Yaskawa INFORM job: DEMO_ROOF_SIDE_0625_3PAINT_47.JBI

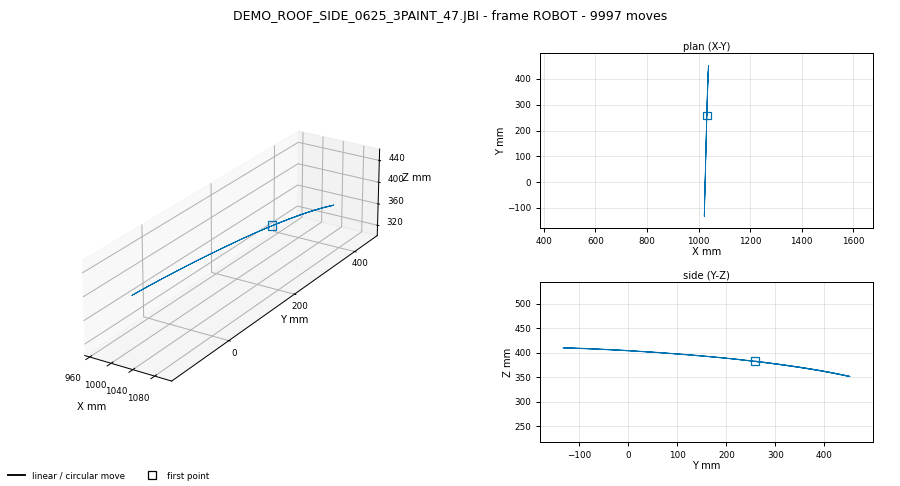
[picture p0: tool path of DEMO_ROOF_SIDE_0625_3PAINT_47.JBI in frame ROBOT, 9997 of 9997 moves have a stored position in this frame; points joined in program order, loops and branches not executed]
/JOB
//NAME DEMO_ROOF_SIDE_0625_3PAINT47
//POS
///NPOS 9997,0,0,0,0,0
///TOOL 0
///USER 0
///POSTYPE ROBOT
///RECTAN
///RCONF 1,0,0,0,0,0,0,0,0,0,0,0,0,0,0,0,0,0,0,0,0,0,0,0
C00000=1032.456,258.256,382.887,170.687,44.569,158.534
C00001=1032.463,258.505,382.858,170.690,44.569,158.534
C00002=1032.469,258.753,382.828,170.693,44.568,158.534
C00003=1032.477,259.001,382.799,170.697,44.568,158.535
C00004=1032.483,259.249,382.770,170.701,44.568,158.535
C00005=1032.490,259.497,382.740,170.704,44.568,158.535
C00006=1032.497,259.745,382.710,170.707,44.567,158.535
C00007=1032.504,259.994,382.681,170.711,44.567,158.536
C00008=1032.510,260.241,382.651,170.714,44.567,158.536
C00009=1032.517,260.490,382.621,170.718,44.567,158.536
C00010=1032.525,260.738,382.592,170.721,44.567,158.537
C00011=1032.531,260.986,382.563,170.725,44.566,158.537
C00012=1032.538,261.234,382.533,170.728,44.566,158.537
C00013=1032.545,261.482,382.503,170.731,44.566,158.537
C00014=1032.552,261.730,382.473,170.734,44.566,158.538
C00015=1032.558,261.979,382.444,170.739,44.566,158.538
C00016=1032.565,262.227,382.414,170.742,44.566,158.538
C00017=1032.572,262.475,382.383,170.745,44.566,158.539
C00018=1032.581,262.826,382.341,170.749,44.566,158.539
C00019=1032.590,263.179,382.299,170.755,44.566,158.540
C00020=1032.600,263.530,382.256,170.759,44.566,158.540
C00021=1032.609,263.882,382.214,170.765,44.566,158.541
C00022=1032.616,264.130,382.183,170.768,44.566,158.541
C00023=1032.623,264.378,382.154,170.771,44.566,158.541
C00024=1032.630,264.626,382.124,170.775,44.566,158.541
C00025=1032.636,264.875,382.093,170.779,44.566,158.542
C00026=1032.643,265.122,382.063,170.782,44.566,158.542
C00027=1032.650,265.370,382.033,170.786,44.566,158.542
C00028=1032.656,265.619,382.003,170.789,44.566,158.543
C00029=1032.662,265.867,381.973,170.792,44.566,158.543
C00030=1032.670,266.115,381.943,170.796,44.565,158.543
C00031=1032.677,266.363,381.913,170.800,44.565,158.544
C00032=1032.683,266.611,381.883,170.803,44.565,158.544
C00033=1032.690,266.859,381.852,170.806,44.565,158.544
C00034=1032.697,267.108,381.822,170.810,44.565,158.545
C00035=1032.703,267.355,381.792,170.814,44.565,158.545
C00036=1032.710,267.604,381.762,170.817,44.565,158.545
C00037=1032.717,267.851,381.731,170.821,44.566,158.546
C00038=1032.723,268.099,381.701,170.824,44.566,158.546
C00039=1032.730,268.347,381.671,170.828,44.565,158.546
C00040=1032.737,268.596,381.640,170.831,44.565,158.547
C00041=1032.743,268.843,381.610,170.835,44.565,158.547
C00042=1032.750,269.092,381.579,170.838,44.565,158.547
C00043=1032.757,269.340,381.549,170.842,44.566,158.548
C00044=1032.764,269.588,381.519,170.846,44.566,158.548
C00045=1032.770,269.835,381.488,170.849,44.566,158.549
C00046=1032.777,270.084,381.458,170.852,44.566,158.549
C00047=1032.784,270.332,381.427,170.856,44.566,158.549
C00048=1032.791,270.580,381.397,170.860,44.566,158.549
C00049=1032.797,270.828,381.366,170.864,44.566,158.550
C00050=1032.804,271.076,381.336,170.867,44.566,158.550
C00051=1032.811,271.324,381.305,170.870,44.566,158.551
C00052=1032.818,271.573,381.275,170.874,44.566,158.551
C00053=1032.824,271.820,381.244,170.878,44.567,158.551
C00054=1032.831,272.068,381.214,170.881,44.566,158.552
C00055=1032.837,272.317,381.183,170.885,44.566,158.552
C00056=1032.844,272.564,381.152,170.889,44.567,158.553
C00057=1032.851,272.812,381.122,170.892,44.567,158.553
C00058=1032.857,273.060,381.091,170.896,44.567,158.553
C00059=1032.865,273.308,381.060,170.900,44.567,158.554
C00060=1032.871,273.557,381.030,170.903,44.567,158.554
C00061=1032.878,273.804,380.998,170.907,44.567,158.554
C00062=1032.884,274.052,380.969,170.910,44.568,158.555
C00063=1032.891,274.300,380.937,170.914,44.568,158.555
C00064=1032.897,274.548,380.906,170.918,44.568,158.555
C00065=1032.905,274.796,380.876,170.921,44.568,158.556
C00066=1032.911,275.045,380.845,170.926,44.568,158.556
C00067=1032.918,275.292,380.813,170.929,44.568,158.557
C00068=1032.925,275.540,380.784,170.932,44.569,158.557
C00069=1032.931,275.788,380.752,170.936,44.569,158.557
C00070=1032.938,276.036,380.721,170.940,44.569,158.558
C00071=1032.945,276.284,380.691,170.943,44.569,158.558
C00072=1032.952,276.532,380.659,170.947,44.569,158.558
C00073=1032.958,276.780,380.628,170.951,44.569,158.559
C00074=1032.969,277.137,380.585,170.957,44.569,158.560
C00075=1032.978,277.493,380.540,170.961,44.570,158.560
C00076=1032.988,277.850,380.495,170.967,44.570,158.561
C00077=1032.997,278.206,380.451,170.972,44.570,158.561
C00078=1033.004,278.453,380.419,170.976,44.571,158.562
C00079=1033.011,278.702,380.388,170.980,44.571,158.562
C00080=1033.017,278.950,380.357,170.984,44.571,158.562
C00081=1033.024,279.198,380.326,170.987,44.571,158.563
C00082=1033.031,279.446,380.294,170.992,44.572,158.563
C00083=1033.037,279.694,380.263,170.995,44.572,158.564
C00084=1033.044,279.942,380.232,170.998,44.572,158.564
C00085=1033.051,280.190,380.201,171.003,44.573,158.565
C00086=1033.058,280.438,380.170,171.006,44.573,158.565
C00087=1033.065,280.686,380.138,171.010,44.573,158.565
C00088=1033.071,280.933,380.107,171.014,44.573,158.566
C00089=1033.078,281.181,380.075,171.018,44.574,158.566
C00090=1033.085,281.429,380.044,171.021,44.574,158.567
C00091=1033.092,281.677,380.013,171.025,44.574,158.567
C00092=1033.098,281.925,379.981,171.029,44.575,158.568
C00093=1033.105,282.173,379.950,171.032,44.575,158.568
C00094=1033.112,282.421,379.918,171.037,44.575,158.568
C00095=1033.119,282.669,379.887,171.040,44.576,158.569
C00096=1033.125,282.917,379.855,171.045,44.575,158.569
C00097=1033.132,283.165,379.824,171.048,44.576,158.570
C00098=1033.139,283.412,379.793,171.052,44.577,158.570
C00099=1033.145,283.660,379.761,171.056,44.576,158.570
C00100=1033.153,283.908,379.730,171.059,44.577,158.571
C00101=1033.160,284.156,379.699,171.064,44.577,158.571
C00102=1033.166,284.404,379.667,171.067,44.578,158.572
C00103=1033.173,284.652,379.636,171.071,44.578,158.572
C00104=1033.180,284.900,379.605,171.075,44.578,158.573
C00105=1033.187,285.147,379.573,171.079,44.579,158.573
C00106=1033.194,285.396,379.541,171.083,44.579,158.574
C00107=1033.201,285.644,379.510,171.087,44.579,158.574
C00108=1033.208,285.891,379.478,171.091,44.580,158.575
C00109=1033.214,286.139,379.446,171.094,44.580,158.575
C00110=1033.221,286.387,379.415,171.098,44.580,158.575
C00111=1033.228,286.635,379.383,171.102,44.581,158.576
C00112=1033.235,286.883,379.352,171.106,44.581,158.576
C00113=1033.241,287.130,379.319,171.111,44.582,158.577
C00114=1033.248,287.379,379.287,171.114,44.582,158.577
C00115=1033.255,287.627,379.256,171.118,44.582,158.578
C00116=1033.262,287.874,379.224,171.122,44.583,158.578
C00117=1033.269,288.122,379.192,171.125,44.583,158.579
C00118=1033.275,288.370,379.161,171.130,44.584,158.579
C00119=1033.282,288.618,379.128,171.133,44.584,158.580
C00120=1033.289,288.866,379.096,171.138,44.585,158.580
C00121=1033.296,289.114,379.064,171.142,44.585,158.581
C00122=1033.303,289.361,379.033,171.146,44.585,158.581
C00123=1033.310,289.609,379.001,171.150,44.586,158.582
C00124=1033.316,289.857,378.969,171.154,44.586,158.582
C00125=1033.322,290.105,378.937,171.157,44.586,158.582
C00126=1033.330,290.353,378.905,171.162,44.587,158.583
C00127=1033.337,290.601,378.873,171.165,44.587,158.583
C00128=1033.343,290.848,378.841,171.170,44.588,158.584
C00129=1033.350,291.096,378.808,171.174,44.588,158.584
C00130=1033.361,291.464,378.761,171.179,44.589,158.585
C00131=1033.371,291.833,378.713,171.185,44.590,158.586
C00132=1033.381,292.202,378.665,171.192,44.591,158.587
C00133=1033.391,292.570,378.617,171.198,44.591,158.587
C00134=1033.398,292.818,378.586,171.201,44.592,158.588
C00135=1033.405,293.066,378.553,171.206,44.592,158.588
C00136=1033.412,293.314,378.521,171.209,44.593,158.589
C00137=1033.418,293.561,378.489,171.214,44.593,158.589
C00138=1033.425,293.810,378.456,171.218,44.595,158.590
C00139=1033.432,294.057,378.424,171.222,44.595,158.590
C00140=1033.439,294.304,378.392,171.226,44.596,158.591
C00141=1033.446,294.553,378.359,171.230,44.596,158.591
C00142=1033.453,294.801,378.327,171.234,44.596,158.592
C00143=1033.459,295.048,378.295,171.238,44.597,158.592
C00144=1033.466,295.296,378.262,171.242,44.598,158.593
C00145=1033.473,295.544,378.229,171.247,44.598,158.594
C00146=1033.479,295.791,378.197,171.250,44.599,158.594
C00147=1033.486,296.039,378.164,171.255,44.599,158.595
C00148=1033.493,296.287,378.131,171.258,44.601,158.595
C00149=1033.500,296.534,378.099,171.263,44.601,158.596
C00150=1033.506,296.782,378.066,171.267,44.601,158.596
C00151=1033.513,297.030,378.033,171.271,44.603,158.597
C00152=1033.520,297.278,378.001,171.276,44.603,158.597
C00153=1033.526,297.525,377.968,171.279,44.604,158.598
C00154=1033.533,297.774,377.935,171.284,44.605,158.599
C00155=1033.540,298.021,377.903,171.288,44.605,158.599
C00156=1033.546,298.268,377.870,171.292,44.606,158.600
C00157=1033.553,298.517,377.837,171.296,44.607,158.600
C00158=1033.560,298.764,377.803,171.300,44.607,158.601
C00159=1033.568,299.012,377.771,171.304,44.608,158.601
C00160=1033.574,299.259,377.738,171.309,44.609,158.602
C00161=1033.580,299.507,377.705,171.313,44.609,158.602
C00162=1033.587,299.755,377.672,171.317,44.610,158.603
C00163=1033.594,300.002,377.640,171.322,44.611,158.603
C00164=1033.601,300.250,377.606,171.325,44.612,158.604
C00165=1033.608,300.498,377.573,171.330,44.612,158.605
C00166=1033.615,300.746,377.541,171.334,44.613,158.605
C00167=1033.621,300.993,377.508,171.338,44.614,158.606
C00168=1033.629,301.241,377.474,171.343,44.614,158.606
C00169=1033.635,301.489,377.442,171.347,44.615,158.607
C00170=1033.643,301.737,377.409,171.351,44.616,158.607
C00171=1033.649,301.983,377.376,171.356,44.617,158.608
C00172=1033.656,302.232,377.343,171.359,44.617,158.609
C00173=1033.662,302.479,377.310,171.364,44.618,158.609
C00174=1033.670,302.727,377.277,171.368,44.619,158.610
C00175=1033.677,302.974,377.244,171.373,44.620,158.610
C00176=1033.684,303.223,377.211,171.377,44.620,158.611
C00177=1033.690,303.470,377.177,171.381,44.622,158.612
C00178=1033.698,303.718,377.145,171.385,44.622,158.612
C00179=1033.705,303.965,377.111,171.390,44.623,158.613
C00180=1033.711,304.213,377.078,171.394,44.623,158.613
C00181=1033.718,304.461,377.044,171.399,44.624,158.614
C00182=1033.725,304.708,377.012,171.403,44.625,158.614
C00183=1033.733,304.955,376.978,171.407,44.626,158.615
C00184=1033.740,305.204,376.945,171.412,44.627,158.616
C00185=1033.746,305.451,376.912,171.416,44.627,158.616
C00186=1033.757,305.836,376.861,171.422,44.629,158.617
C00187=1033.768,306.222,376.808,171.429,44.630,158.618
C00188=1033.779,306.608,376.757,171.436,44.631,158.619
C00189=1033.791,306.993,376.705,171.443,44.632,158.620
C00190=1033.798,307.241,376.672,171.448,44.633,158.621
C00191=1033.804,307.488,376.638,171.452,44.634,158.621
C00192=1033.811,307.736,376.605,171.456,44.635,158.622
C00193=1033.818,307.984,376.572,171.461,44.636,158.623
C00194=1033.826,308.231,376.538,171.465,44.637,158.623
C00195=1033.833,308.478,376.505,171.470,44.638,158.624
C00196=1033.840,308.726,376.471,171.474,44.638,158.624
C00197=1033.847,308.974,376.438,171.479,44.639,158.625
C00198=1033.855,309.222,376.405,171.483,44.641,158.626
C00199=1033.861,309.469,376.371,171.487,44.641,158.626
C00200=1033.869,309.716,376.337,171.492,44.642,158.627
C00201=1033.876,309.964,376.304,171.497,44.643,158.628
C00202=1033.883,310.212,376.270,171.502,44.644,158.628
C00203=1033.891,310.460,376.237,171.505,44.644,158.629
C00204=1033.898,310.707,376.203,171.510,44.645,158.629
C00205=1033.904,310.954,376.170,171.515,44.646,158.630
C00206=1033.912,311.202,376.136,171.520,44.647,158.631
C00207=1033.919,311.450,376.102,171.524,44.648,158.631
C00208=1033.926,311.697,376.068,171.528,44.650,158.632
C00209=1033.933,311.945,376.035,171.533,44.651,158.633
C00210=1033.939,312.192,376.001,171.538,44.651,158.633
C00211=1033.946,312.440,375.967,171.542,44.653,158.634
C00212=1033.953,312.688,375.933,171.546,44.654,158.635
C00213=1033.960,312.935,375.898,171.551,44.655,158.635
C00214=1033.967,313.183,375.864,171.556,44.656,158.636
C00215=1033.973,313.430,375.830,171.560,44.657,158.637
C00216=1033.981,313.678,375.796,171.565,44.658,158.637
C00217=1033.988,313.925,375.762,171.569,44.659,158.638
C00218=1033.994,314.173,375.727,171.574,44.660,158.639
C00219=1034.002,314.420,375.693,171.579,44.661,158.640
C00220=1034.008,314.668,375.659,171.583,44.663,158.640
C00221=1034.016,314.915,375.624,171.588,44.663,158.641
C00222=1034.022,315.162,375.591,171.593,44.664,158.642
C00223=1034.029,315.410,375.556,171.597,44.665,158.642
C00224=1034.036,315.657,375.522,171.602,44.667,158.643
C00225=1034.043,315.905,375.488,171.606,44.668,158.644
C00226=1034.050,316.152,375.453,171.611,44.669,158.645
C00227=1034.057,316.400,375.419,171.616,44.670,158.645
C00228=1034.064,316.648,375.385,171.621,44.671,158.646
C00229=1034.071,316.895,375.350,171.626,44.673,158.647
C00230=1034.078,317.143,375.316,171.629,44.674,158.647
C00231=1034.085,317.390,375.281,171.634,44.675,158.648
C00232=1034.092,317.638,375.247,171.639,44.676,158.649
C00233=1034.099,317.885,375.212,171.644,44.677,158.650
C00234=1034.106,318.133,375.178,171.649,44.678,158.650
C00235=1034.113,318.380,375.143,171.654,44.679,158.651
C00236=1034.120,318.628,375.110,171.659,44.681,158.652
C00237=1034.127,318.875,375.074,171.662,44.682,158.652
C00238=1034.135,319.122,375.040,171.667,44.683,158.653
C00239=1034.141,319.370,375.005,171.672,44.685,158.654
C00240=1034.149,319.617,374.971,171.677,44.686,158.655
C00241=1034.157,319.866,374.937,171.682,44.687,158.655
C00242=1034.167,320.256,374.882,171.689,44.689,158.657
C00243=1034.179,320.646,374.827,171.697,44.691,158.658
C00244=1034.189,321.036,374.773,171.705,44.692,158.659
C00245=1034.201,321.427,374.718,171.713,44.695,158.660
C00246=1034.209,321.674,374.683,171.717,44.696,158.661
C00247=1034.215,321.922,374.649,171.722,44.697,158.662
C00248=1034.223,322.169,374.614,171.727,44.698,158.662
C00249=1034.230,322.417,374.579,171.731,44.700,158.663
C00250=1034.238,322.664,374.544,171.736,44.701,158.664
C00251=1034.244,322.911,374.509,171.741,44.702,158.665
C00252=1034.252,323.158,374.475,171.746,44.703,158.665
C00253=1034.259,323.407,374.440,171.751,44.705,158.666
C00254=1034.266,323.654,374.405,171.756,44.706,158.667
C00255=1034.273,323.901,374.370,171.761,44.707,158.668
C00256=1034.281,324.149,374.335,171.766,44.708,158.669
C00257=1034.288,324.396,374.300,171.771,44.710,158.669
C00258=1034.296,324.643,374.265,171.775,44.711,158.670
C00259=1034.303,324.892,374.230,171.780,44.712,158.671
C00260=1034.310,325.139,374.195,171.785,44.714,158.672
C00261=1034.317,325.386,374.160,171.790,44.715,158.672
C00262=1034.325,325.634,374.125,171.795,44.717,158.673
C00263=1034.332,325.881,374.090,171.800,44.718,158.674
C00264=1034.340,326.128,374.056,171.805,44.719,158.675
C00265=1034.347,326.376,374.020,171.810,44.721,158.676
C00266=1034.354,326.623,373.986,171.815,44.722,158.676
C00267=1034.362,326.870,373.950,171.820,44.723,158.677
C00268=1034.370,327.118,373.915,171.826,44.724,158.678
C00269=1034.376,327.365,373.880,171.831,44.726,158.679
C00270=1034.385,327.613,373.845,171.836,44.727,158.680
C00271=1034.391,327.860,373.810,171.841,44.729,158.681
C00272=1034.399,328.108,373.775,171.846,44.730,158.681
C00273=1034.406,328.355,373.739,171.851,44.732,158.682
C00274=1034.414,328.603,373.703,171.856,44.733,158.683
C00275=1034.421,328.850,373.668,171.861,44.734,158.684
C00276=1034.428,329.097,373.633,171.866,44.736,158.685
C00277=1034.436,329.345,373.598,171.871,44.737,158.686
C00278=1034.443,329.591,373.562,171.876,44.739,158.686
C00279=1034.450,329.839,373.526,171.881,44.740,158.687
C00280=1034.457,330.086,373.490,171.886,44.742,158.688
C00281=1034.465,330.334,373.455,171.891,44.744,158.689
C00282=1034.472,330.581,373.419,171.896,44.745,158.690
C00283=1034.479,330.829,373.384,171.901,44.747,158.691
C00284=1034.486,331.076,373.348,171.906,44.748,158.691
C00285=1034.494,331.324,373.312,171.912,44.750,158.692
C00286=1034.501,331.571,373.276,171.917,44.751,158.693
C00287=1034.508,331.818,373.240,171.922,44.753,158.694
C00288=1034.515,332.065,373.205,171.928,44.755,158.695
C00289=1034.524,332.313,373.169,171.933,44.756,158.696
C00290=1034.530,332.560,373.134,171.938,44.758,158.697
C00291=1034.538,332.807,373.098,171.943,44.759,158.698
C00292=1034.546,333.055,373.062,171.948,44.761,158.699
C00293=1034.553,333.302,373.026,171.954,44.762,158.699
C00294=1034.560,333.550,372.990,171.959,44.764,158.700
C00295=1034.567,333.796,372.955,171.964,44.766,158.701
C00296=1034.575,334.044,372.918,171.969,44.768,158.702
C00297=1034.583,334.291,372.882,171.974,44.769,158.703
C00298=1034.594,334.678,372.826,171.983,44.772,158.705
C00299=1034.605,335.063,372.770,171.991,44.774,158.706
C00300=1034.617,335.448,372.714,172.000,44.777,158.707
C00301=1034.628,335.834,372.657,172.008,44.780,158.709
C00302=1034.635,336.082,372.620,172.013,44.781,158.710
C00303=1034.642,336.329,372.585,172.018,44.783,158.711
C00304=1034.650,336.576,372.548,172.024,44.785,158.712
C00305=1034.658,336.823,372.512,172.029,44.786,158.712
C00306=1034.665,337.070,372.476,172.034,44.788,158.713
C00307=1034.672,337.318,372.439,172.039,44.790,158.714
C00308=1034.679,337.565,372.403,172.045,44.792,158.715
C00309=1034.687,337.813,372.367,172.051,44.793,158.716
C00310=1034.695,338.060,372.330,172.056,44.796,158.717
C00311=1034.702,338.306,372.294,172.061,44.797,158.718
C00312=1034.709,338.554,372.257,172.066,44.799,158.719
C00313=1034.717,338.802,372.221,172.073,44.801,158.720
C00314=1034.724,339.049,372.185,172.078,44.803,158.721
C00315=1034.732,339.296,372.148,172.083,44.804,158.722
C00316=1034.740,339.543,372.112,172.088,44.806,158.723
C00317=1034.746,339.790,372.075,172.095,44.808,158.724
C00318=1034.754,340.037,372.038,172.100,44.810,158.725
C00319=1034.762,340.285,372.002,172.105,44.812,158.726
C00320=1034.770,340.532,371.966,172.111,44.813,158.727
C00321=1034.778,340.779,371.929,172.116,44.815,158.728
C00322=1034.785,341.027,371.892,172.122,44.818,158.729
C00323=1034.793,341.273,371.855,172.127,44.820,158.730
C00324=1034.799,341.521,371.819,172.133,44.821,158.731
C00325=1034.807,341.767,371.782,172.138,44.823,158.732
C00326=1034.815,342.015,371.746,172.144,44.825,158.733
C00327=1034.822,342.262,371.708,172.150,44.827,158.734
C00328=1034.830,342.509,371.672,172.155,44.829,158.735
C00329=1034.837,342.756,371.634,172.160,44.831,158.736
C00330=1034.845,343.003,371.598,172.167,44.833,158.737
C00331=1034.852,343.251,371.561,172.172,44.835,158.738
C00332=1034.860,343.498,371.524,172.177,44.837,158.739
C00333=1034.867,343.745,371.486,172.184,44.839,158.740
C00334=1034.875,343.992,371.450,172.189,44.841,158.741
C00335=1034.882,344.240,371.413,172.194,44.843,158.742
C00336=1034.890,344.486,371.376,172.200,44.845,158.743
C00337=1034.897,344.734,371.338,172.206,44.847,158.744
C00338=1034.905,344.981,371.302,172.211,44.849,158.745
C00339=1034.912,345.228,371.264,172.217,44.851,158.746
C00340=1034.920,345.475,371.227,172.223,44.853,158.747
C00341=1034.927,345.722,371.190,172.228,44.855,158.748
C00342=1034.935,345.969,371.153,172.234,44.857,158.749
C00343=1034.942,346.216,371.115,172.240,44.859,158.750
C00344=1034.951,346.464,371.078,172.246,44.861,158.752
C00345=1034.958,346.711,371.041,172.251,44.863,158.753
C00346=1034.966,346.958,371.003,172.257,44.866,158.754
C00347=1034.974,347.205,370.966,172.263,44.867,158.755
C00348=1034.981,347.452,370.929,172.269,44.870,158.756
C00349=1034.989,347.699,370.892,172.275,44.872,158.757
C00350=1034.997,347.946,370.854,172.280,44.874,158.758
C00351=1035.005,348.193,370.817,172.287,44.876,158.759
C00352=1035.012,348.440,370.779,172.292,44.878,158.760
C00353=1035.019,348.688,370.742,172.298,44.881,158.761
C00354=1035.032,349.070,370.684,172.308,44.884,158.763
C00355=1035.043,349.452,370.625,172.316,44.887,158.765
C00356=1035.055,349.835,370.568,172.325,44.891,158.766
C00357=1035.067,350.217,370.509,172.334,44.894,158.768
C00358=1035.075,350.464,370.471,172.341,44.896,158.769
C00359=1035.082,350.711,370.434,172.346,44.899,158.771
C00360=1035.090,350.957,370.396,172.352,44.901,158.772
C00361=1035.098,351.205,370.358,172.358,44.904,158.773
C00362=1035.105,351.452,370.320,172.364,44.905,158.774
C00363=1035.113,351.699,370.282,172.370,44.908,158.775
C00364=1035.121,351.946,370.244,172.376,44.910,158.776
C00365=1035.128,352.193,370.206,172.382,44.913,158.777
C00366=1035.136,352.440,370.168,172.388,44.915,158.778
C00367=1035.144,352.687,370.131,172.395,44.917,158.780
C00368=1035.152,352.934,370.092,172.400,44.920,158.781
C00369=1035.159,353.180,370.054,172.407,44.922,158.782
C00370=1035.167,353.428,370.016,172.412,44.924,158.783
C00371=1035.175,353.675,369.978,172.419,44.926,158.784
C00372=1035.184,353.922,369.940,172.424,44.929,158.785
C00373=1035.191,354.169,369.902,172.431,44.931,158.787
C00374=1035.199,354.416,369.864,172.437,44.934,158.788
C00375=1035.207,354.663,369.826,172.443,44.936,158.789
C00376=1035.214,354.910,369.788,172.449,44.938,158.790
C00377=1035.222,355.157,369.749,172.455,44.941,158.791
C00378=1035.230,355.404,369.711,172.461,44.944,158.793
C00379=1035.238,355.650,369.673,172.468,44.945,158.794
C00380=1035.247,355.898,369.635,172.473,44.948,158.795
C00381=1035.254,356.144,369.596,172.480,44.951,158.796
C00382=1035.262,356.391,369.558,172.487,44.953,158.798
C00383=1035.270,356.638,369.519,172.492,44.956,158.799
C00384=1035.277,356.885,369.480,172.499,44.958,158.800
C00385=1035.285,357.132,369.442,172.505,44.961,158.801
C00386=1035.293,357.379,369.403,172.511,44.963,158.802
C00387=1035.301,357.626,369.365,172.518,44.966,158.804
C00388=1035.309,357.873,369.327,172.524,44.968,158.805
C00389=1035.317,358.120,369.288,172.530,44.971,158.806
C00390=1035.324,358.366,369.250,172.536,44.973,158.807
C00391=1035.333,358.614,369.211,172.543,44.976,158.809
C00392=1035.341,358.861,369.172,172.549,44.978,158.810
C00393=1035.349,359.107,369.133,172.555,44.981,158.811
C00394=1035.357,359.354,369.095,172.562,44.983,158.812
C00395=1035.365,359.601,369.056,172.569,44.986,158.814
C00396=1035.372,359.848,369.018,172.574,44.989,158.815
C00397=1035.381,360.094,368.979,172.581,44.992,158.816
C00398=1035.389,360.342,368.940,172.587,44.994,158.818
C00399=1035.396,360.588,368.901,172.594,44.997,158.819
C00400=1035.404,360.835,368.862,172.600,45.000,158.820
C00401=1035.412,361.082,368.823,172.606,45.002,158.821
C00402=1035.421,361.329,368.784,172.613,45.005,158.823
C00403=1035.428,361.575,368.746,172.620,45.008,158.824
C00404=1035.436,361.822,368.706,172.627,45.010,158.825
C00405=1035.444,362.069,368.667,172.632,45.013,158.827
C00406=1035.453,362.316,368.628,172.639,45.016,158.828
C00407=1035.460,362.563,368.588,172.646,45.019,158.830
C00408=1035.468,362.809,368.550,172.652,45.021,158.831
C00409=1035.476,363.056,368.510,172.659,45.024,158.832
C00410=1035.488,363.445,368.448,172.669,45.029,158.834
C00411=1035.502,363.833,368.386,172.680,45.033,158.836
C00412=1035.514,364.222,368.325,172.690,45.038,158.839
C00413=1035.527,364.610,368.262,172.700,45.042,158.841
C00414=1035.534,364.857,368.222,172.707,45.045,158.842
C00415=1035.543,365.104,368.184,172.714,45.048,158.844
C00416=1035.551,365.351,368.144,172.721,45.050,158.845
C00417=1035.559,365.597,368.105,172.728,45.053,158.846
C00418=1035.567,365.844,368.065,172.734,45.056,158.848
C00419=1035.575,366.091,368.025,172.741,45.059,158.849
C00420=1035.583,366.338,367.986,172.747,45.062,158.850
C00421=1035.592,366.584,367.947,172.754,45.065,158.852
C00422=1035.600,366.831,367.907,172.761,45.068,158.853
C00423=1035.608,367.078,367.867,172.768,45.071,158.855
C00424=1035.616,367.324,367.827,172.774,45.074,158.856
C00425=1035.625,367.570,367.787,172.781,45.077,158.858
C00426=1035.633,367.817,367.748,172.788,45.080,158.859
C00427=1035.641,368.064,367.708,172.795,45.083,158.860
C00428=1035.649,368.311,367.669,172.802,45.086,158.862
C00429=1035.658,368.558,367.628,172.809,45.089,158.863
C00430=1035.666,368.804,367.589,172.816,45.092,158.865
C00431=1035.675,369.051,367.549,172.823,45.095,158.866
C00432=1035.682,369.298,367.509,172.829,45.098,158.868
C00433=1035.691,369.544,367.469,172.836,45.101,158.869
C00434=1035.699,369.791,367.429,172.843,45.104,158.870
C00435=1035.708,370.037,367.389,172.850,45.107,158.872
C00436=1035.716,370.284,367.349,172.857,45.110,158.873
C00437=1035.724,370.530,367.308,172.864,45.113,158.875
C00438=1035.732,370.777,367.268,172.872,45.116,158.876
C00439=1035.741,371.023,367.228,172.879,45.119,158.878
C00440=1035.748,371.270,367.189,172.886,45.123,158.880
C00441=1035.757,371.517,367.147,172.893,45.126,158.881
C00442=1035.765,371.763,367.107,172.900,45.129,158.882
C00443=1035.773,372.010,367.068,172.907,45.132,158.884
C00444=1035.781,372.256,367.027,172.914,45.135,158.885
C00445=1035.790,372.503,366.986,172.921,45.139,158.887
C00446=1035.798,372.750,366.945,172.928,45.142,158.889
C00447=1035.807,372.996,366.905,172.935,45.145,158.890
C00448=1035.815,373.243,366.865,172.943,45.148,158.892
C00449=1035.823,373.489,366.824,172.950,45.152,158.893
C00450=1035.831,373.736,366.784,172.957,45.155,158.895
C00451=1035.841,373.982,366.743,172.964,45.158,158.896
C00452=1035.849,374.229,366.703,172.971,45.162,158.898
C00453=1035.857,374.476,366.662,172.978,45.165,158.899
C00454=1035.865,374.722,366.621,172.986,45.168,158.901
C00455=1035.874,374.968,366.581,172.994,45.172,158.903
C00456=1035.883,375.215,366.540,173.001,45.175,158.904
C00457=1035.891,375.461,366.499,173.008,45.178,158.906
C00458=1035.899,375.708,366.458,173.015,45.182,158.907
C00459=1035.908,375.954,366.418,173.023,45.185,158.909
C00460=1035.917,376.201,366.377,173.030,45.188,158.911
C00461=1035.925,376.447,366.336,173.037,45.192,158.912
C00462=1035.934,376.694,366.295,173.045,45.195,158.914
C00463=1035.942,376.940,366.254,173.052,45.198,158.915
C00464=1035.951,377.187,366.214,173.060,45.202,158.917
C00465=1035.960,377.433,366.172,173.067,45.205,158.919
C00466=1035.974,377.842,366.105,173.079,45.211,158.921
C00467=1035.988,378.251,366.036,173.092,45.217,158.924
C00468=1036.002,378.660,365.968,173.105,45.223,158.927
C00469=1036.016,379.069,365.900,173.117,45.229,158.930
C00470=1036.025,379.315,365.858,173.125,45.232,158.931
C00471=1036.033,379.562,365.817,173.132,45.236,158.933
C00472=1036.041,379.808,365.775,173.140,45.239,158.935
C00473=1036.050,380.055,365.733,173.147,45.243,158.937
C00474=1036.059,380.300,365.692,173.156,45.247,158.938
C00475=1036.067,380.547,365.651,173.163,45.250,158.940
C00476=1036.076,380.794,365.609,173.170,45.254,158.942
C00477=1036.085,381.040,365.567,173.178,45.257,158.943
C00478=1036.094,381.286,365.526,173.186,45.262,158.945
C00479=1036.102,381.532,365.484,173.194,45.265,158.947
C00480=1036.111,381.779,365.442,173.202,45.269,158.949
C00481=1036.119,382.026,365.401,173.210,45.272,158.950
C00482=1036.128,382.272,365.359,173.217,45.276,158.952
C00483=1036.137,382.518,365.318,173.224,45.280,158.954
C00484=1036.146,382.764,365.276,173.233,45.284,158.956
C00485=1036.154,383.010,365.234,173.240,45.287,158.957
C00486=1036.164,383.256,365.192,173.248,45.291,158.959
C00487=1036.173,383.503,365.150,173.257,45.295,158.961
C00488=1036.181,383.749,365.108,173.264,45.298,158.963
C00489=1036.190,383.996,365.066,173.273,45.302,158.964
C00490=1036.199,384.242,365.025,173.280,45.306,158.966
C00491=1036.208,384.488,364.983,173.289,45.310,158.968
C00492=1036.217,384.734,364.940,173.296,45.314,158.970
C00493=1036.226,384.980,364.899,173.304,45.317,158.972
C00494=1036.235,385.227,364.857,173.312,45.322,158.973
C00495=1036.243,385.473,364.814,173.320,45.325,158.975
C00496=1036.252,385.719,364.772,173.329,45.329,158.977
C00497=1036.261,385.966,364.731,173.336,45.333,158.979
C00498=1036.270,386.211,364.688,173.345,45.337,158.981
C00499=1036.279,386.458,364.646,173.353,45.341,158.983
C00500=1036.289,386.703,364.604,173.360,45.345,158.985
C00501=1036.297,386.950,364.562,173.369,45.349,158.986
C00502=1036.306,387.196,364.519,173.377,45.353,158.988
C00503=1036.315,387.443,364.477,173.385,45.357,158.990
C00504=1036.325,387.689,364.435,173.394,45.361,158.992
C00505=1036.333,387.935,364.392,173.402,45.365,158.994
C00506=1036.342,388.181,364.350,173.410,45.369,158.996
C00507=1036.351,388.427,364.308,173.418,45.373,158.998
C00508=1036.360,388.673,364.264,173.427,45.377,159.000
C00509=1036.370,388.919,364.222,173.435,45.381,159.002
C00510=1036.378,389.165,364.179,173.443,45.386,159.004
C00511=1036.387,389.411,364.136,173.452,45.389,159.006
C00512=1036.396,389.657,364.093,173.460,45.394,159.008
C00513=1036.406,389.904,364.050,173.469,45.398,159.009
C00514=1036.415,390.149,364.008,173.478,45.402,159.012
C00515=1036.424,390.395,363.965,173.485,45.406,159.013
C00516=1036.433,390.642,363.922,173.494,45.410,159.015
C00517=1036.442,390.888,363.879,173.503,45.415,159.017
C00518=1036.451,391.134,363.837,173.511,45.419,159.019
C00519=1036.460,391.380,363.793,173.520,45.423,159.021
C00520=1036.469,391.626,363.750,173.529,45.427,159.023
C00521=1036.478,391.872,363.707,173.536,45.432,159.025
C00522=1036.489,392.155,363.658,173.546,45.437,159.028
C00523=1036.499,392.436,363.608,173.556,45.441,159.030
C00524=1036.509,392.719,363.559,173.567,45.447,159.032
C00525=1036.521,393.001,363.509,173.576,45.452,159.035
C00526=1036.530,393.246,363.465,173.585,45.456,159.037
C00527=1036.539,393.493,363.422,173.593,45.460,159.039
C00528=1036.548,393.738,363.379,173.602,45.465,159.041
C00529=1036.557,393.985,363.335,173.611,45.469,159.043
C00530=1036.573,394.392,363.263,173.626,45.476,159.046
C00531=1036.588,394.800,363.192,173.640,45.484,159.050
C00532=1036.604,395.207,363.119,173.655,45.491,159.053
C00533=1036.619,395.614,363.047,173.670,45.499,159.057
C00534=1036.629,395.860,363.003,173.679,45.503,159.059
C00535=1036.638,396.106,362.959,173.688,45.508,159.061
C00536=1036.647,396.352,362.915,173.697,45.512,159.063
C00537=1036.657,396.597,362.872,173.706,45.517,159.066
C00538=1036.666,396.844,362.828,173.715,45.521,159.068
C00539=1036.675,397.089,362.784,173.724,45.526,159.070
C00540=1036.685,397.335,362.740,173.733,45.530,159.072
C00541=1036.694,397.581,362.696,173.742,45.535,159.074
C00542=1036.704,397.827,362.652,173.751,45.540,159.076
C00543=1036.714,398.073,362.608,173.760,45.544,159.079
C00544=1036.722,398.319,362.564,173.769,45.549,159.081
C00545=1036.732,398.564,362.520,173.779,45.554,159.083
C00546=1036.741,398.810,362.476,173.788,45.558,159.085
C00547=1036.752,399.056,362.432,173.797,45.563,159.087
C00548=1036.761,399.302,362.388,173.806,45.568,159.090
C00549=1036.771,399.548,362.343,173.816,45.573,159.092
C00550=1036.780,399.794,362.299,173.826,45.577,159.094
C00551=1036.790,400.039,362.254,173.835,45.582,159.097
C00552=1036.799,400.286,362.210,173.844,45.587,159.099
C00553=1036.809,400.531,362.165,173.854,45.592,159.101
C00554=1036.818,400.777,362.121,173.863,45.597,159.103
C00555=1036.828,401.023,362.076,173.872,45.602,159.106
C00556=1036.837,401.269,362.032,173.882,45.606,159.108
C00557=1036.847,401.514,361.987,173.891,45.612,159.110
C00558=1036.857,401.760,361.943,173.901,45.616,159.113
C00559=1036.867,402.005,361.898,173.911,45.621,159.115
C00560=1036.876,402.252,361.854,173.920,45.626,159.117
C00561=1036.886,402.497,361.809,173.930,45.631,159.120
C00562=1036.896,402.743,361.764,173.939,45.636,159.122
C00563=1036.906,402.989,361.719,173.949,45.641,159.124
C00564=1036.916,403.234,361.674,173.959,45.646,159.127
C00565=1036.924,403.480,361.628,173.968,45.651,159.129
C00566=1036.934,403.726,361.584,173.978,45.656,159.132
C00567=1036.945,403.972,361.538,173.988,45.661,159.134
C00568=1036.954,404.217,361.494,173.998,45.666,159.136
C00569=1036.964,404.463,361.449,174.007,45.672,159.139
C00570=1036.973,404.708,361.403,174.018,45.677,159.141
C00571=1036.984,404.954,361.358,174.027,45.682,159.144
C00572=1036.993,405.200,361.313,174.037,45.687,159.146
C00573=1037.003,405.445,361.267,174.047,45.692,159.149
C00574=1037.013,405.691,361.221,174.057,45.697,159.151
C00575=1037.023,405.937,361.177,174.066,45.703,159.154
C00576=1037.033,406.182,361.131,174.077,45.708,159.156
C00577=1037.043,406.428,361.086,174.087,45.713,159.159
C00578=1037.053,406.660,361.043,174.097,45.718,159.161
C00579=1037.061,406.892,361.000,174.106,45.723,159.163
C00580=1037.071,407.123,360.956,174.116,45.728,159.166
C00581=1037.080,407.356,360.913,174.125,45.733,159.168
C00582=1037.090,407.588,360.870,174.135,45.738,159.171
C00583=1037.099,407.820,360.827,174.144,45.743,159.173
C00584=1037.110,408.051,360.784,174.154,45.748,159.175
C00585=1037.118,408.283,360.741,174.164,45.754,159.178
C00586=1037.129,408.528,360.695,174.174,45.759,159.180
C00587=1037.139,408.775,360.649,174.185,45.764,159.183
C00588=1037.149,409.020,360.604,174.195,45.769,159.185
C00589=1037.159,409.265,360.558,174.205,45.775,159.188
C00590=1037.169,409.511,360.511,174.215,45.780,159.191
C00591=1037.179,409.756,360.466,174.226,45.786,159.193
C00592=1037.190,410.002,360.420,174.237,45.791,159.196
C00593=1037.200,410.247,360.374,174.247,45.797,159.199
C00594=1037.210,410.493,360.327,174.258,45.802,159.201
C00595=1037.221,410.739,360.282,174.269,45.808,159.204
C00596=1037.232,410.985,360.236,174.279,45.814,159.207
C00597=1037.241,411.229,360.189,174.289,45.819,159.209
C00598=1037.252,411.475,360.143,174.300,45.824,159.212
C00599=1037.262,411.721,360.096,174.310,45.830,159.215
C00600=1037.273,411.966,360.050,174.321,45.836,159.217
C00601=1037.283,412.211,360.003,174.332,45.842,159.220
C00602=1037.293,412.457,359.956,174.343,45.847,159.223
C00603=1037.303,412.702,359.910,174.354,45.853,159.226
C00604=1037.314,412.948,359.863,174.364,45.859,159.228
C00605=1037.324,413.193,359.817,174.375,45.865,159.231
C00606=1037.334,413.439,359.770,174.387,45.870,159.234
C00607=1037.345,413.684,359.723,174.398,45.876,159.237
C00608=1037.355,413.929,359.677,174.409,45.882,159.240
C00609=1037.365,414.175,359.629,174.420,45.887,159.242
C00610=1037.376,414.420,359.583,174.431,45.894,159.245
C00611=1037.386,414.665,359.536,174.442,45.900,159.248
C00612=1037.397,414.911,359.488,174.452,45.905,159.251
C00613=1037.408,415.156,359.441,174.464,45.911,159.254
C00614=1037.418,415.401,359.394,174.476,45.917,159.257
C00615=1037.429,415.646,359.347,174.486,45.923,159.259
C00616=1037.439,415.891,359.300,174.497,45.929,159.262
C00617=1037.450,416.137,359.253,174.509,45.935,159.265
C00618=1037.461,416.382,359.206,174.520,45.941,159.268
C00619=1037.471,416.628,359.159,174.531,45.947,159.271
C00620=1037.482,416.874,359.111,174.544,45.953,159.274
C00621=1037.493,417.119,359.065,174.555,45.959,159.277
C00622=1037.504,417.364,359.016,174.566,45.965,159.280
C00623=1037.514,417.609,358.969,174.578,45.971,159.283
C00624=1037.525,417.855,358.922,174.589,45.978,159.286
C00625=1037.536,418.100,358.874,174.601,45.983,159.289
C00626=1037.547,418.344,358.826,174.613,45.990,159.292
C00627=1037.558,418.590,358.779,174.625,45.996,159.295
C00628=1037.568,418.835,358.731,174.636,46.002,159.298
C00629=1037.579,419.080,358.683,174.647,46.009,159.301
C00630=1037.590,419.326,358.635,174.659,46.015,159.304
C00631=1037.601,419.571,358.587,174.671,46.021,159.307
C00632=1037.611,419.816,358.539,174.683,46.027,159.310
C00633=1037.622,420.061,358.491,174.695,46.034,159.313
C00634=1037.633,420.306,358.443,174.706,46.040,159.316
C00635=1037.644,420.551,358.395,174.719,46.046,159.320
C00636=1037.655,420.796,358.346,174.731,46.052,159.323
C00637=1037.666,421.042,358.298,174.742,46.059,159.326
C00638=1037.677,421.278,358.252,174.755,46.065,159.329
C00639=1037.688,421.514,358.206,174.766,46.071,159.332
C00640=1037.697,421.750,358.159,174.778,46.078,159.335
C00641=1037.709,421.986,358.113,174.789,46.084,159.338
C00642=1037.720,422.223,358.066,174.802,46.090,159.341
C00643=1037.730,422.459,358.019,174.813,46.097,159.344
C00644=1037.741,422.695,357.973,174.825,46.102,159.347
C00645=1037.752,422.932,357.925,174.837,46.109,159.350
C00646=1037.763,423.177,357.877,174.849,46.116,159.354
C00647=1037.775,423.421,357.829,174.862,46.122,159.357
C00648=1037.786,423.667,357.780,174.875,46.129,159.360
C00649=1037.797,423.912,357.731,174.887,46.135,159.363
C00650=1037.808,424.157,357.683,174.900,46.142,159.367
C00651=1037.819,424.402,357.634,174.912,46.149,159.370
C00652=1037.831,424.647,357.584,174.925,46.155,159.373
C00653=1037.842,424.891,357.535,174.938,46.162,159.377
C00654=1037.853,425.136,357.486,174.950,46.169,159.380
C00655=1037.865,425.381,357.437,174.963,46.176,159.384
C00656=1037.875,425.627,357.389,174.976,46.182,159.387
C00657=1037.887,425.871,357.339,174.988,46.189,159.390
C00658=1037.898,426.115,357.290,175.001,46.196,159.394
C00659=1037.910,426.361,357.240,175.014,46.203,159.397
C00660=1037.922,426.606,357.191,175.027,46.210,159.401
C00661=1037.933,426.850,357.142,175.041,46.217,159.404
C00662=1037.944,427.095,357.093,175.054,46.224,159.408
C00663=1037.956,427.340,357.043,175.066,46.231,159.411
C00664=1037.967,427.585,356.994,175.080,46.238,159.415
C00665=1037.979,427.830,356.945,175.093,46.244,159.418
C00666=1037.991,428.074,356.895,175.106,46.252,159.422
C00667=1038.002,428.320,356.845,175.119,46.259,159.425
C00668=1038.014,428.564,356.795,175.133,46.266,159.429
C00669=1038.025,428.809,356.745,175.146,46.273,159.432
C00670=1038.037,429.054,356.696,175.159,46.280,159.436
C00671=1038.049,429.298,356.645,175.173,46.287,159.439
C00672=1038.060,429.543,356.595,175.186,46.294,159.443
C00673=1038.072,429.788,356.545,175.200,46.301,159.447
C00674=1038.083,430.032,356.495,175.214,46.309,159.450
C00675=1038.095,430.277,356.445,175.228,46.316,159.454
C00676=1038.107,430.522,356.394,175.241,46.323,159.458
C00677=1038.119,430.766,356.344,175.255,46.330,159.461
C00678=1038.131,431.011,356.294,175.268,46.338,159.465
C00679=1038.143,431.256,356.243,175.283,46.345,159.469
C00680=1038.154,431.500,356.194,175.297,46.353,159.473
C00681=1038.166,431.745,356.142,175.310,46.360,159.476
C00682=1038.179,431.990,356.092,175.324,46.367,159.480
C00683=1038.191,432.234,356.042,175.339,46.375,159.484
C00684=1038.202,432.478,355.991,175.353,46.382,159.488
C00685=1038.214,432.723,355.941,175.366,46.390,159.491
C00686=1038.226,432.967,355.890,175.381,46.397,159.495
C00687=1038.239,433.212,355.839,175.395,46.404,159.499
C00688=1038.250,433.457,355.788,175.410,46.412,159.503
C00689=1038.263,433.701,355.737,175.424,46.419,159.507
C00690=1038.275,433.946,355.687,175.439,46.427,159.511
C00691=1038.287,434.190,355.636,175.453,46.435,159.515
C00692=1038.300,434.435,355.585,175.468,46.442,159.519
C00693=1038.312,434.679,355.534,175.482,46.450,159.523
C00694=1038.324,434.923,355.483,175.497,46.458,159.526
C00695=1038.336,435.168,355.431,175.512,46.466,159.530
C00696=1038.349,435.412,355.380,175.526,46.473,159.534
C00697=1038.361,435.657,355.329,175.541,46.481,159.538
C00698=1038.373,435.897,355.279,175.555,46.489,159.542
C00699=1038.385,436.137,355.227,175.570,46.496,159.546
C00700=1038.398,436.377,355.177,175.585,46.504,159.550
C00701=1038.409,436.617,355.127,175.599,46.512,159.554
C00702=1038.422,436.857,355.076,175.614,46.519,159.558
C00703=1038.435,437.097,355.025,175.630,46.527,159.562
C00704=1038.447,437.337,354.974,175.644,46.535,159.567
C00705=1038.459,437.576,354.923,175.659,46.543,159.571
C00706=1038.471,437.821,354.871,175.674,46.551,159.575
C00707=1038.484,438.065,354.819,175.690,46.559,159.579
C00708=1038.497,438.310,354.767,175.705,46.567,159.583
C00709=1038.509,438.553,354.715,175.721,46.575,159.587
C00710=1038.522,438.798,354.663,175.736,46.583,159.591
C00711=1038.534,439.042,354.611,175.752,46.591,159.596
C00712=1038.548,439.286,354.559,175.767,46.599,159.600
C00713=1038.560,439.530,354.507,175.783,46.607,159.604
C00714=1038.573,439.775,354.454,175.798,46.616,159.609
C00715=1038.586,440.019,354.402,175.814,46.624,159.613
C00716=1038.599,440.263,354.350,175.830,46.632,159.617
C00717=1038.612,440.507,354.297,175.847,46.640,159.622
C00718=1038.624,440.751,354.244,175.862,46.648,159.626
C00719=1038.638,440.995,354.191,175.878,46.657,159.631
C00720=1038.650,441.239,354.139,175.894,46.665,159.635
C00721=1038.663,441.483,354.086,175.911,46.673,159.639
C00722=1038.676,441.727,354.033,175.927,46.682,159.644
C00723=1038.689,441.972,353.980,175.943,46.690,159.648
C00724=1038.703,442.215,353.928,175.960,46.699,159.653
C00725=1038.716,442.459,353.874,175.976,46.707,159.657
C00726=1038.729,442.703,353.821,175.993,46.716,159.662
C00727=1038.742,442.947,353.768,176.009,46.724,159.666
C00728=1038.755,443.191,353.715,176.026,46.733,159.671
C00729=1038.768,443.435,353.662,176.042,46.741,159.676
C00730=1038.781,443.679,353.608,176.059,46.750,159.680
C00731=1038.795,443.923,353.556,176.076,46.759,159.685
C00732=1038.808,444.166,353.502,176.092,46.767,159.689
C00733=1038.821,444.410,353.449,176.110,46.776,159.694
C00734=1038.835,444.653,353.396,176.126,46.784,159.699
C00735=1038.850,444.896,353.344,176.144,46.793,159.703
C00736=1038.865,445.140,353.291,176.160,46.801,159.708
C00737=1038.880,445.384,353.239,176.178,46.810,159.713
C00738=1038.896,445.627,353.188,176.196,46.818,159.717
C00739=1038.912,445.871,353.138,176.212,46.826,159.722
C00740=1038.929,446.114,353.088,176.229,46.834,159.726
C00741=1038.947,446.359,353.038,176.248,46.842,159.731
C00742=1038.966,446.602,352.989,176.265,46.850,159.736
C00743=1038.984,446.846,352.939,176.283,46.857,159.740
C00744=1039.004,447.091,352.891,176.301,46.865,159.745
C00745=1039.024,447.335,352.843,176.318,46.872,159.749
C00746=1039.045,447.580,352.796,176.336,46.880,159.754
C00747=1039.066,447.824,352.748,176.355,46.887,159.758
C00748=1039.087,448.068,352.701,176.372,46.894,159.762
C00749=1039.109,448.313,352.656,176.390,46.901,159.767
C00750=1039.132,448.558,352.610,176.409,46.908,159.771
C00751=1039.156,448.803,352.564,176.427,46.915,159.776
C00752=1039.180,449.048,352.520,176.445,46.923,159.780
C00753=1039.204,449.292,352.475,176.464,46.929,159.785
C00754=1039.229,449.538,352.431,176.482,46.936,159.789
C00755=1039.255,449.782,352.388,176.501,46.942,159.793
C00756=1039.280,450.028,352.345,176.520,46.949,159.798
C00757=1039.307,450.273,352.302,176.539,46.955,159.802
C00758=1039.354,450.687,352.232,176.571,46.966,159.809
C00759=1039.402,451.102,352.162,176.603,46.976,159.817
C00760=1039.452,451.515,352.094,176.635,46.986,159.824
C00761=1039.502,451.927,352.028,176.668,46.996,159.831
C00762=1039.208,451.977,351.708,176.671,47.071,159.854
C00763=1039.158,451.579,351.772,176.640,47.061,159.847
C00764=1039.110,451.180,351.837,176.608,47.052,159.840
C00765=1039.064,450.780,351.904,176.577,47.042,159.833
C00766=1039.019,450.380,351.972,176.546,47.032,159.826
C00767=1038.991,450.136,352.014,176.527,47.025,159.822
C00768=1038.965,449.890,352.057,176.508,47.019,159.817
C00769=1038.939,449.645,352.100,176.489,47.012,159.813
C00770=1038.913,449.400,352.143,176.470,47.006,159.809
C00771=1038.889,449.155,352.187,176.452,46.999,159.804
C00772=1038.864,448.910,352.232,176.433,46.993,159.800
C00773=1038.841,448.665,352.277,176.415,46.986,159.795
C00774=1038.818,448.421,352.323,176.397,46.979,159.791
C00775=1038.795,448.175,352.369,176.378,46.972,159.786
C00776=1038.773,447.931,352.415,176.359,46.965,159.782
C00777=1038.752,447.686,352.462,176.342,46.957,159.778
C00778=1038.731,447.442,352.509,176.324,46.950,159.773
C00779=1038.710,447.197,352.557,176.306,46.943,159.769
C00780=1038.691,446.953,352.606,176.289,46.935,159.764
C00781=1038.671,446.709,352.653,176.270,46.928,159.760
C00782=1038.653,446.465,352.703,176.253,46.920,159.755
C00783=1038.634,446.221,352.753,176.235,46.912,159.750
C00784=1038.617,445.977,352.803,176.217,46.905,159.746
C00785=1038.600,445.734,352.853,176.200,46.897,159.741
C00786=1038.584,445.490,352.904,176.183,46.888,159.737
C00787=1038.568,445.246,352.956,176.165,46.880,159.732
C00788=1038.553,445.002,353.007,176.148,46.872,159.728
C00789=1038.539,444.760,353.060,176.131,46.864,159.723
C00790=1038.524,444.516,353.112,176.114,46.856,159.718
C00791=1038.511,444.273,353.165,176.097,46.847,159.714
C00792=1038.497,444.029,353.219,176.080,46.838,159.709
C00793=1038.483,443.786,353.272,176.063,46.830,159.704
C00794=1038.471,443.543,353.325,176.046,46.821,159.700
C00795=1038.457,443.298,353.378,176.030,46.813,159.695
C00796=1038.444,443.054,353.432,176.013,46.804,159.691
C00797=1038.431,442.810,353.485,175.996,46.796,159.686
C00798=1038.417,442.567,353.537,175.979,46.788,159.681
C00799=1038.404,442.323,353.591,175.963,46.779,159.677
C00800=1038.391,442.079,353.644,175.946,46.771,159.672
C00801=1038.378,441.835,353.697,175.930,46.763,159.668
C00802=1038.366,441.591,353.749,175.914,46.754,159.663
C00803=1038.353,441.347,353.802,175.897,46.746,159.659
C00804=1038.339,441.103,353.855,175.882,46.737,159.655
C00805=1038.326,440.859,353.907,175.866,46.729,159.650
C00806=1038.313,440.615,353.961,175.849,46.721,159.646
C00807=1038.301,440.371,354.013,175.833,46.713,159.641
C00808=1038.288,440.127,354.066,175.817,46.705,159.637
C00809=1038.275,439.882,354.118,175.802,46.696,159.633
C00810=1038.261,439.638,354.170,175.786,46.688,159.628
C00811=1038.249,439.394,354.222,175.770,46.680,159.624
C00812=1038.236,439.149,354.275,175.755,46.672,159.620
C00813=1038.224,438.906,354.327,175.739,46.664,159.615
C00814=1038.211,438.661,354.379,175.722,46.656,159.611
C00815=1038.198,438.417,354.431,175.708,46.648,159.607
C00816=1038.186,438.173,354.484,175.692,46.640,159.603
C00817=1038.173,437.929,354.535,175.677,46.632,159.599
C00818=1038.160,437.685,354.588,175.661,46.625,159.594
C00819=1038.148,437.444,354.638,175.646,46.617,159.590
C00820=1038.136,437.203,354.690,175.631,46.609,159.586
C00821=1038.123,436.963,354.741,175.616,46.601,159.582
C00822=1038.111,436.722,354.791,175.601,46.593,159.578
C00823=1038.098,436.481,354.842,175.586,46.586,159.574
C00824=1038.086,436.241,354.893,175.571,46.578,159.570
C00825=1038.075,436.000,354.944,175.557,46.571,159.566
C00826=1038.062,435.759,354.995,175.542,46.563,159.562
C00827=1038.049,435.514,355.046,175.527,46.555,159.558
C00828=1038.037,435.270,355.097,175.513,46.548,159.554
C00829=1038.025,435.025,355.149,175.498,46.540,159.550
C00830=1038.013,434.781,355.199,175.483,46.532,159.546
C00831=1038.001,434.537,355.251,175.468,46.524,159.542
C00832=1037.988,434.292,355.302,175.453,46.517,159.538
C00833=1037.976,434.048,355.352,175.439,46.510,159.534
C00834=1037.964,433.804,355.404,175.424,46.502,159.530
C00835=1037.951,433.559,355.454,175.410,46.495,159.527
C00836=1037.940,433.314,355.505,175.395,46.487,159.523
C00837=1037.927,433.070,355.556,175.381,46.480,159.519
C00838=1037.915,432.825,355.606,175.368,46.472,159.515
C00839=1037.903,432.581,355.658,175.353,46.465,159.511
C00840=1037.890,432.336,355.708,175.339,46.458,159.508
C00841=1037.879,432.091,355.759,175.325,46.450,159.504
C00842=1037.866,431.847,355.809,175.310,46.443,159.500
C00843=1037.855,431.603,355.859,175.297,46.436,159.496
C00844=1037.843,431.358,355.910,175.283,46.428,159.492
C00845=1037.830,431.113,355.960,175.268,46.421,159.489
C00846=1037.819,430.868,356.011,175.254,46.414,159.485
C00847=1037.807,430.624,356.061,175.241,46.406,159.481
C00848=1037.795,430.379,356.111,175.227,46.400,159.478
C00849=1037.784,430.135,356.161,175.214,46.392,159.474
C00850=1037.772,429.890,356.211,175.200,46.385,159.470
C00851=1037.760,429.645,356.262,175.186,46.378,159.467
C00852=1037.748,429.401,356.312,175.172,46.371,159.463
C00853=1037.736,429.156,356.362,175.159,46.364,159.459
C00854=1037.725,428.911,356.412,175.145,46.357,159.456
C00855=1037.714,428.667,356.461,175.132,46.350,159.452
C00856=1037.702,428.421,356.512,175.118,46.343,159.448
C00857=1037.690,428.177,356.562,175.105,46.336,159.445
C00858=1037.678,427.932,356.611,175.092,46.329,159.441
C00859=1037.667,427.687,356.661,175.078,46.322,159.438
C00860=1037.655,427.442,356.711,175.065,46.315,159.434
C00861=1037.644,427.197,356.760,175.052,46.308,159.431
C00862=1037.632,426.953,356.809,175.038,46.301,159.427
C00863=1037.621,426.707,356.859,175.026,46.294,159.424
C00864=1037.609,426.463,356.908,175.013,46.287,159.421
C00865=1037.598,426.218,356.957,175.000,46.281,159.417
C00866=1037.587,425.973,357.007,174.986,46.274,159.414
C00867=1037.575,425.728,357.056,174.974,46.267,159.410
C00868=1037.563,425.483,357.105,174.961,46.261,159.407
C00869=1037.552,425.238,357.154,174.948,46.254,159.404
C00870=1037.541,424.993,357.204,174.935,46.247,159.400
C00871=1037.530,424.748,357.253,174.923,46.240,159.397
C00872=1037.518,424.504,357.302,174.910,46.233,159.393
C00873=1037.507,424.258,357.350,174.897,46.227,159.390
C00874=1037.496,424.014,357.399,174.885,46.220,159.387
C00875=1037.484,423.769,357.448,174.872,46.213,159.383
C00876=1037.473,423.524,357.496,174.859,46.207,159.380
C00877=1037.462,423.279,357.545,174.847,46.201,159.377
C00878=1037.451,423.033,357.593,174.834,46.194,159.374
C00879=1037.440,422.796,357.641,174.822,46.188,159.371
C00880=1037.430,422.559,357.687,174.811,46.182,159.368
C00881=1037.419,422.321,357.735,174.798,46.176,159.364
C00882=1037.407,422.085,357.781,174.787,46.169,159.361
C00883=1037.397,421.847,357.828,174.775,46.163,159.358
C00884=1037.386,421.610,357.875,174.763,46.157,159.355
C00885=1037.375,421.372,357.922,174.751,46.151,159.352
C00886=1037.365,421.135,357.969,174.740,46.144,159.349
C00887=1037.354,420.890,358.017,174.727,46.138,159.346
C00888=1037.342,420.645,358.065,174.715,46.132,159.343
C00889=1037.331,420.400,358.113,174.703,46.126,159.340
C00890=1037.320,420.155,358.161,174.691,46.119,159.336
C00891=1037.309,419.910,358.209,174.679,46.113,159.333
C00892=1037.299,419.665,358.257,174.668,46.107,159.330
C00893=1037.288,419.419,358.305,174.655,46.101,159.327
C00894=1037.277,419.174,358.353,174.643,46.094,159.324
C00895=1037.266,418.929,358.401,174.632,46.088,159.321
C00896=1037.255,418.684,358.449,174.620,46.082,159.318
C00897=1037.245,418.438,358.497,174.608,46.076,159.315
C00898=1037.233,418.193,358.544,174.596,46.070,159.312
C00899=1037.223,417.948,358.592,174.585,46.064,159.309
C00900=1037.213,417.703,358.639,174.573,46.058,159.306
C00901=1037.202,417.457,358.687,174.562,46.051,159.303
C00902=1037.191,417.213,358.735,174.550,46.046,159.300
C00903=1037.180,416.967,358.782,174.539,46.040,159.297
C00904=1037.170,416.722,358.829,174.528,46.033,159.294
C00905=1037.159,416.476,358.876,174.515,46.028,159.291
C00906=1037.148,416.231,358.923,174.504,46.022,159.288
C00907=1037.137,415.986,358.971,174.494,46.016,159.286
C00908=1037.126,415.741,359.018,174.482,46.010,159.283
C00909=1037.116,415.495,359.066,174.470,46.004,159.280
C00910=1037.105,415.250,359.113,174.459,45.998,159.277
C00911=1037.094,415.005,359.159,174.448,45.993,159.274
C00912=1037.084,414.760,359.207,174.437,45.987,159.271
C00913=1037.074,414.514,359.253,174.426,45.981,159.268
C00914=1037.063,414.268,359.300,174.415,45.975,159.265
C00915=1037.053,414.023,359.347,174.404,45.969,159.263
C00916=1037.042,413.778,359.394,174.392,45.963,159.260
C00917=1037.032,413.532,359.441,174.381,45.958,159.257
C00918=1037.022,413.287,359.488,174.370,45.952,159.254
C00919=1037.011,413.042,359.534,174.359,45.946,159.251
C00920=1037.001,412.796,359.581,174.349,45.940,159.249
C00921=1036.990,412.551,359.627,174.338,45.935,159.246
C00922=1036.980,412.305,359.675,174.327,45.929,159.243
C00923=1036.970,412.060,359.721,174.316,45.924,159.240
C00924=1036.959,411.815,359.768,174.305,45.918,159.238
C00925=1036.949,411.569,359.814,174.295,45.913,159.235
C00926=1036.939,411.324,359.860,174.284,45.907,159.232
C00927=1036.929,411.078,359.906,174.273,45.901,159.230
C00928=1036.918,410.833,359.953,174.262,45.896,159.227
C00929=1036.908,410.587,359.999,174.252,45.890,159.224
C00930=1036.898,410.341,360.045,174.241,45.885,159.222
C00931=1036.887,410.096,360.091,174.231,45.879,159.219
C00932=1036.876,409.850,360.137,174.220,45.874,159.216
C00933=1036.866,409.605,360.183,174.209,45.869,159.214
C00934=1036.857,409.359,360.229,174.199,45.863,159.211
C00935=1036.846,409.114,360.275,174.188,45.858,159.208
C00936=1036.835,408.868,360.321,174.179,45.853,159.206
C00937=1036.825,408.623,360.366,174.168,45.847,159.203
C00938=1036.816,408.377,360.412,174.158,45.842,159.201
C00939=1036.806,408.144,360.455,174.148,45.837,159.198
C00940=1036.796,407.911,360.499,174.138,45.832,159.196
C00941=1036.787,407.679,360.543,174.128,45.827,159.193
C00942=1036.777,407.445,360.586,174.118,45.822,159.191
C00943=1036.768,407.212,360.629,174.109,45.817,159.189
C00944=1036.758,406.979,360.672,174.099,45.812,159.186
C00945=1036.749,406.746,360.715,174.089,45.807,159.184
C00946=1036.739,406.513,360.759,174.080,45.802,159.181
C00947=1036.729,406.267,360.804,174.069,45.797,159.179
C00948=1036.719,406.022,360.849,174.060,45.791,159.176
C00949=1036.709,405.776,360.895,174.050,45.787,159.174
C00950=1036.699,405.531,360.941,174.039,45.782,159.171
C00951=1036.689,405.285,360.986,174.030,45.776,159.169
C00952=1036.679,405.039,361.031,174.020,45.771,159.166
C00953=1036.670,404.794,361.077,174.010,45.766,159.164
C00954=1036.660,404.548,361.122,174.000,45.761,159.161
C00955=1036.650,404.302,361.167,173.990,45.756,159.159
C00956=1036.640,404.057,361.212,173.980,45.751,159.157
C00957=1036.631,403.811,361.257,173.970,45.746,159.154
C00958=1036.621,403.565,361.303,173.961,45.741,159.152
C00959=1036.611,403.320,361.348,173.950,45.736,159.149
C00960=1036.601,403.074,361.393,173.941,45.731,159.147
C00961=1036.592,402.829,361.437,173.932,45.726,159.145
C00962=1036.582,402.583,361.482,173.922,45.721,159.142
C00963=1036.572,402.336,361.527,173.912,45.716,159.140
C00964=1036.563,402.091,361.572,173.902,45.711,159.138
C00965=1036.553,401.845,361.617,173.893,45.706,159.135
C00966=1036.544,401.600,361.662,173.883,45.701,159.133
C00967=1036.534,401.353,361.706,173.874,45.697,159.131
C00968=1036.524,401.108,361.751,173.865,45.692,159.128
C00969=1036.515,400.862,361.796,173.854,45.687,159.126
C00970=1036.505,400.616,361.840,173.845,45.682,159.124
C00971=1036.496,400.371,361.885,173.836,45.677,159.122
C00972=1036.485,400.125,361.928,173.826,45.673,159.119
C00973=1036.476,399.879,361.973,173.817,45.668,159.117
C00974=1036.466,399.633,362.017,173.808,45.663,159.115
C00975=1036.457,399.388,362.062,173.798,45.658,159.112
C00976=1036.447,399.142,362.106,173.789,45.654,159.110
C00977=1036.438,398.895,362.150,173.780,45.649,159.108
C00978=1036.428,398.650,362.195,173.771,45.644,159.106
C00979=1036.418,398.404,362.238,173.761,45.640,159.103
C00980=1036.408,398.158,362.282,173.752,45.635,159.101
C00981=1036.400,397.913,362.326,173.743,45.631,159.099
C00982=1036.390,397.666,362.370,173.734,45.626,159.097
C00983=1036.381,397.420,362.414,173.724,45.621,159.095
C00984=1036.370,397.175,362.459,173.715,45.617,159.092
C00985=1036.362,396.930,362.502,173.706,45.612,159.090
C00986=1036.352,396.684,362.546,173.697,45.608,159.088
C00987=1036.343,396.437,362.591,173.688,45.603,159.086
C00988=1036.333,396.192,362.634,173.679,45.598,159.084
C00989=1036.324,395.946,362.677,173.670,45.594,159.082
C00990=1036.315,395.699,362.721,173.661,45.590,159.080
C00991=1036.305,395.453,362.765,173.651,45.585,159.077
C00992=1036.297,395.208,362.809,173.642,45.581,159.075
C00993=1036.286,394.962,362.853,173.634,45.577,159.073
C00994=1036.278,394.717,362.896,173.625,45.572,159.071
C00995=1036.268,394.470,362.940,173.616,45.568,159.069
C00996=1036.258,394.224,362.983,173.607,45.563,159.067
C00997=1036.250,393.978,363.026,173.598,45.559,159.065
C00998=1036.240,393.732,363.070,173.589,45.554,159.063
C00999=1036.232,393.509,363.109,173.582,45.550,159.061
C01000=1036.224,393.286,363.149,173.573,45.547,159.059
C01001=1036.215,393.063,363.187,173.566,45.543,159.057
C01002=1036.207,392.840,363.227,173.557,45.539,159.055
C01003=1036.198,392.618,363.266,173.550,45.535,159.054
C01004=1036.190,392.395,363.306,173.542,45.531,159.052
C01005=1036.182,392.172,363.344,173.534,45.528,159.050
C01006=1036.174,391.949,363.384,173.526,45.524,159.048
C01007=1036.164,391.703,363.426,173.518,45.519,159.046
C01008=1036.155,391.456,363.470,173.509,45.515,159.044
C01009=1036.146,391.211,363.513,173.500,45.511,159.042
C01010=1036.137,390.965,363.556,173.492,45.507,159.040
C01011=1036.127,390.719,363.599,173.484,45.503,159.038
C01012=1036.119,390.473,363.642,173.475,45.498,159.036
C01013=1036.110,390.227,363.684,173.467,45.494,159.034
C01014=1036.100,389.980,363.727,173.458,45.490,159.032
C01015=1036.091,389.734,363.770,173.449,45.486,159.030
C01016=1036.083,389.488,363.813,173.441,45.482,159.028
C01017=1036.073,389.242,363.856,173.433,45.478,159.026
C01018=1036.064,388.996,363.898,173.424,45.474,159.024
C01019=1036.055,388.750,363.941,173.416,45.470,159.022
C01020=1036.046,388.504,363.984,173.407,45.466,159.020
C01021=1036.037,388.257,364.026,173.399,45.462,159.018
C01022=1036.028,388.011,364.069,173.391,45.458,159.017
C01023=1036.019,387.766,364.111,173.383,45.454,159.015
C01024=1036.010,387.519,364.154,173.374,45.450,159.013
C01025=1036.001,387.273,364.196,173.366,45.446,159.011
C01026=1035.992,387.027,364.238,173.358,45.442,159.009
C01027=1035.982,386.780,364.280,173.350,45.438,159.007
C01028=1035.974,386.534,364.323,173.341,45.434,159.005
C01029=1035.965,386.288,364.365,173.334,45.430,159.004
C01030=1035.956,386.042,364.408,173.325,45.427,159.002
C01031=1035.947,385.796,364.449,173.317,45.423,159.000
C01032=1035.938,385.550,364.492,173.309,45.419,158.998
C01033=1035.929,385.304,364.533,173.301,45.415,158.996
C01034=1035.920,385.057,364.575,173.292,45.411,158.994
C01035=1035.911,384.811,364.618,173.285,45.408,158.993
C01036=1035.902,384.565,364.660,173.277,45.404,158.991
C01037=1035.893,384.319,364.702,173.268,45.400,158.989
C01038=1035.884,384.072,364.743,173.261,45.396,158.987
C01039=1035.875,383.826,364.785,173.252,45.393,158.985
C01040=1035.866,383.580,364.828,173.245,45.389,158.983
C01041=1035.857,383.334,364.869,173.237,45.385,158.982
C01042=1035.848,383.087,364.911,173.229,45.381,158.980
C01043=1035.840,382.841,364.953,173.221,45.377,158.978
C01044=1035.831,382.594,364.995,173.214,45.374,158.976
C01045=1035.823,382.349,365.036,173.205,45.370,158.975
C01046=1035.814,382.102,365.078,173.198,45.367,158.973
C01047=1035.804,381.821,365.126,173.188,45.362,158.971
C01048=1035.794,381.540,365.173,173.180,45.358,158.969
C01049=1035.784,381.258,365.221,173.171,45.354,158.967
C01050=1035.775,380.977,365.268,173.162,45.350,158.965
C01051=1035.766,380.731,365.310,173.154,45.346,158.963
C01052=1035.757,380.484,365.351,173.147,45.343,158.962
C01053=1035.748,380.239,365.393,173.139,45.340,158.960
C01054=1035.739,379.992,365.434,173.131,45.335,158.958
C01055=1035.731,379.745,365.475,173.123,45.332,158.956
C01056=1035.723,379.499,365.517,173.116,45.329,158.955
C01057=1035.714,379.253,365.559,173.108,45.325,158.953
C01058=1035.706,379.006,365.600,173.100,45.322,158.951
C01059=1035.693,378.631,365.662,173.089,45.316,158.949
C01060=1035.680,378.254,365.726,173.077,45.311,158.946
C01061=1035.667,377.877,365.789,173.066,45.306,158.944
C01062=1035.654,377.502,365.851,173.055,45.301,158.941
C01063=1035.645,377.255,365.892,173.047,45.297,158.940
C01064=1035.636,377.008,365.933,173.039,45.294,158.938
C01065=1035.627,376.763,365.974,173.032,45.290,158.936
C01066=1035.619,376.516,366.015,173.024,45.287,158.935
C01067=1035.611,376.269,366.056,173.017,45.283,158.933
C01068=1035.601,376.023,366.096,173.010,45.280,158.932
C01069=1035.593,375.776,366.137,173.002,45.277,158.930
C01070=1035.584,375.530,366.179,172.995,45.274,158.928
C01071=1035.576,375.284,366.219,172.988,45.271,158.927
C01072=1035.568,375.037,366.260,172.981,45.267,158.925
C01073=1035.559,374.791,366.300,172.972,45.264,158.923
C01074=1035.551,374.544,366.341,172.965,45.261,158.922
C01075=1035.542,374.297,366.382,172.958,45.257,158.920
C01076=1035.534,374.051,366.423,172.951,45.254,158.919
C01077=1035.525,373.805,366.463,172.943,45.251,158.917
C01078=1035.517,373.558,366.504,172.936,45.248,158.916
C01079=1035.509,373.311,366.543,172.929,45.244,158.914
C01080=1035.500,373.064,366.585,172.922,45.241,158.913
C01081=1035.492,372.818,366.625,172.915,45.238,158.911
C01082=1035.484,372.572,366.665,172.908,45.235,158.910
C01083=1035.475,372.325,366.706,172.900,45.232,158.908
C01084=1035.467,372.078,366.746,172.893,45.229,158.907
C01085=1035.459,371.832,366.786,172.886,45.226,158.905
C01086=1035.450,371.586,366.827,172.879,45.222,158.903
C01087=1035.442,371.339,366.868,172.872,45.219,158.902
C01088=1035.434,371.092,366.908,172.865,45.216,158.901
C01089=1035.425,370.846,366.948,172.858,45.213,158.899
C01090=1035.418,370.599,366.988,172.851,45.210,158.897
C01091=1035.410,370.353,367.028,172.844,45.207,158.896
C01092=1035.401,370.106,367.068,172.836,45.204,158.894
C01093=1035.393,369.859,367.109,172.829,45.201,158.893
C01094=1035.385,369.612,367.149,172.822,45.198,158.892
C01095=1035.376,369.366,367.189,172.816,45.195,158.890
C01096=1035.368,369.120,367.228,172.809,45.192,158.889
C01097=1035.359,368.872,367.268,172.802,45.189,158.887
C01098=1035.351,368.626,367.308,172.795,45.186,158.886
C01099=1035.343,368.379,367.348,172.788,45.183,158.884
C01100=1035.334,368.133,367.387,172.781,45.180,158.883
C01101=1035.327,367.886,367.427,172.774,45.177,158.881
C01102=1035.318,367.639,367.467,172.767,45.174,158.880
C01103=1035.309,367.393,367.507,172.760,45.171,158.879
C01104=1035.302,367.146,367.547,172.753,45.168,158.877
C01105=1035.293,366.900,367.586,172.747,45.166,158.876
C01106=1035.285,366.653,367.626,172.740,45.163,158.874
C01107=1035.277,366.406,367.665,172.733,45.160,158.873
C01108=1035.269,366.160,367.705,172.726,45.157,158.871
C01109=1035.261,365.913,367.744,172.720,45.154,158.870
C01110=1035.252,365.666,367.784,172.713,45.151,158.869
C01111=1035.245,365.419,367.824,172.706,45.148,158.867
C01112=1035.236,365.173,367.863,172.699,45.146,158.866
C01113=1035.228,364.926,367.902,172.692,45.143,158.865
C01114=1035.220,364.679,367.942,172.685,45.140,158.863
C01115=1035.207,364.288,368.005,172.676,45.135,158.861
C01116=1035.195,363.898,368.067,172.665,45.131,158.859
C01117=1035.182,363.508,368.129,172.654,45.127,158.857
C01118=1035.169,363.116,368.191,172.643,45.123,158.855
C01119=1035.161,362.870,368.230,172.638,45.120,158.853
C01120=1035.153,362.624,368.269,172.631,45.117,158.852
C01121=1035.146,362.376,368.309,172.624,45.114,158.851
C01122=1035.137,362.130,368.348,172.617,45.111,158.849
C01123=1035.129,361.883,368.387,172.611,45.109,158.848
C01124=1035.121,361.636,368.427,172.604,45.106,158.847
C01125=1035.113,361.390,368.465,172.598,45.103,158.845
C01126=1035.105,361.143,368.504,172.592,45.101,158.844
C01127=1035.097,360.895,368.543,172.585,45.098,158.843
C01128=1035.089,360.649,368.582,172.578,45.096,158.842
C01129=1035.082,360.402,368.621,172.571,45.093,158.840
C01130=1035.073,360.155,368.660,172.566,45.090,158.839
C01131=1035.065,359.908,368.699,172.559,45.088,158.838
C01132=1035.058,359.662,368.737,172.553,45.085,158.836
C01133=1035.049,359.415,368.776,172.546,45.083,158.835
C01134=1035.041,359.168,368.815,172.540,45.080,158.834
C01135=1035.033,358.921,368.854,172.534,45.078,158.833
C01136=1035.025,358.674,368.892,172.527,45.076,158.831
C01137=1035.017,358.427,368.930,172.520,45.073,158.830
C01138=1035.009,358.181,368.969,172.515,45.070,158.829
C01139=1035.001,357.934,369.008,172.508,45.068,158.828
C01140=1034.993,357.686,369.047,172.502,45.066,158.826
C01141=1034.986,357.440,369.085,172.495,45.063,158.825
C01142=1034.978,357.192,369.124,172.489,45.060,158.824
C01143=1034.971,356.946,369.162,172.483,45.058,158.823
C01144=1034.962,356.699,369.201,172.476,45.056,158.821
C01145=1034.954,356.451,369.239,172.471,45.053,158.820
C01146=1034.947,356.205,369.278,172.464,45.050,158.819
C01147=1034.939,355.958,369.316,172.457,45.048,158.818
C01148=1034.931,355.711,369.355,172.452,45.046,158.817
C01149=1034.923,355.464,369.393,172.445,45.043,158.815
C01150=1034.915,355.217,369.430,172.439,45.041,158.814
C01151=1034.907,354.970,369.469,172.434,45.039,158.813
C01152=1034.899,354.723,369.507,172.427,45.036,158.812
C01153=1034.891,354.476,369.546,172.420,45.034,158.810
C01154=1034.884,354.229,369.583,172.415,45.032,158.809
C01155=1034.876,353.982,369.622,172.408,45.029,158.808
C01156=1034.867,353.736,369.659,172.402,45.027,158.807
C01157=1034.860,353.489,369.698,172.396,45.025,158.806
C01158=1034.852,353.241,369.736,172.390,45.022,158.805
C01159=1034.844,352.995,369.774,172.384,45.020,158.804
C01160=1034.837,352.747,369.812,172.378,45.018,158.802
C01161=1034.829,352.500,369.850,172.372,45.016,158.801
C01162=1034.821,352.254,369.887,172.366,45.013,158.800
C01163=1034.813,352.006,369.925,172.360,45.011,158.799
C01164=1034.805,351.760,369.964,172.354,45.009,158.798
C01165=1034.798,351.513,370.001,172.348,45.007,158.797
C01166=1034.790,351.265,370.039,172.342,45.004,158.795
C01167=1034.783,351.018,370.077,172.336,45.002,158.794
C01168=1034.775,350.772,370.114,172.329,45.000,158.793
C01169=1034.767,350.524,370.153,172.324,44.998,158.792
C01170=1034.759,350.277,370.190,172.317,44.996,158.791
C01171=1034.747,349.894,370.249,172.308,44.992,158.789
C01172=1034.736,349.509,370.308,172.299,44.989,158.787
C01173=1034.724,349.125,370.366,172.290,44.986,158.786
C01174=1034.712,348.740,370.425,172.281,44.982,158.784
C01175=1034.704,348.493,370.462,172.275,44.980,158.783
C01176=1034.696,348.246,370.500,172.269,44.978,158.782
C01177=1034.688,347.999,370.537,172.263,44.976,158.781
C01178=1034.681,347.751,370.575,172.257,44.974,158.780
C01179=1034.673,347.504,370.612,172.252,44.972,158.778
C01180=1034.665,347.257,370.649,172.245,44.970,158.777
C01181=1034.658,347.010,370.687,172.240,44.968,158.776
C01182=1034.650,346.763,370.724,172.234,44.966,158.775
C01183=1034.643,346.516,370.761,172.228,44.964,158.774
C01184=1034.635,346.269,370.798,172.223,44.962,158.773
C01185=1034.627,346.021,370.836,172.217,44.960,158.772
C01186=1034.619,345.775,370.873,172.211,44.958,158.771
C01187=1034.612,345.528,370.910,172.205,44.956,158.770
C01188=1034.605,345.280,370.948,172.200,44.954,158.769
C01189=1034.597,345.033,370.984,172.193,44.952,158.768
C01190=1034.590,344.786,371.022,172.188,44.950,158.767
C01191=1034.582,344.539,371.059,172.183,44.947,158.766
C01192=1034.574,344.292,371.096,172.176,44.946,158.765
C01193=1034.566,344.045,371.133,172.171,44.943,158.764
C01194=1034.560,343.797,371.170,172.166,44.941,158.763
C01195=1034.552,343.550,371.207,172.160,44.940,158.762
C01196=1034.544,343.304,371.244,172.154,44.938,158.761
C01197=1034.537,343.056,371.281,172.148,44.936,158.760
C01198=1034.529,342.809,371.317,172.143,44.934,158.759
C01199=1034.521,342.562,371.355,172.137,44.932,158.758
C01200=1034.514,342.314,371.391,172.131,44.931,158.757
C01201=1034.506,342.067,371.429,172.126,44.928,158.756
C01202=1034.499,341.820,371.465,172.121,44.926,158.755
C01203=1034.492,341.573,371.502,172.114,44.924,158.753
C01204=1034.484,341.326,371.538,172.109,44.923,158.753
C01205=1034.477,341.079,371.575,172.104,44.921,158.752
C01206=1034.470,340.831,371.612,172.098,44.919,158.751
C01207=1034.462,340.585,371.649,172.092,44.917,158.750
C01208=1034.454,340.337,371.685,172.087,44.915,158.749
C01209=1034.446,340.090,371.721,172.081,44.914,158.748
C01210=1034.439,339.843,371.759,172.076,44.912,158.747
C01211=1034.431,339.595,371.795,172.071,44.910,158.746
C01212=1034.424,339.348,371.831,172.065,44.908,158.745
C01213=1034.416,339.102,371.868,172.059,44.907,158.744
C01214=1034.409,338.854,371.904,172.054,44.905,158.743
C01215=1034.402,338.606,371.941,172.049,44.903,158.742
C01216=1034.394,338.359,371.977,172.043,44.901,158.741
C01217=1034.386,338.111,372.013,172.038,44.900,158.740
C01218=1034.379,337.865,372.050,172.032,44.898,158.739
C01219=1034.371,337.618,372.086,172.027,44.896,158.738
C01220=1034.364,337.370,372.123,172.021,44.895,158.737
C01221=1034.357,337.123,372.159,172.016,44.893,158.736
C01222=1034.350,336.876,372.195,172.011,44.891,158.735
C01223=1034.342,336.628,372.231,172.006,44.890,158.734
C01224=1034.334,336.381,372.268,171.999,44.888,158.733
C01225=1034.328,336.134,372.304,171.994,44.886,158.733
C01226=1034.320,335.887,372.340,171.989,44.885,158.732
C01227=1034.308,335.499,372.397,171.980,44.882,158.730
C01228=1034.297,335.112,372.454,171.972,44.879,158.729
C01229=1034.286,334.724,372.511,171.964,44.877,158.727
C01230=1034.274,334.335,372.567,171.956,44.874,158.726
C01231=1034.266,334.089,372.602,171.951,44.872,158.725
C01232=1034.259,333.841,372.639,171.945,44.871,158.724
C01233=1034.251,333.594,372.675,171.940,44.870,158.723
C01234=1034.244,333.346,372.710,171.935,44.868,158.722
C01235=1034.237,333.099,372.746,171.930,44.867,158.722
C01236=1034.229,332.851,372.782,171.925,44.865,158.721
C01237=1034.222,332.604,372.818,171.918,44.863,158.720
C01238=1034.215,332.357,372.854,171.913,44.862,158.719
C01239=1034.208,332.110,372.890,171.908,44.860,158.718
C01240=1034.200,331.862,372.925,171.903,44.858,158.717
C01241=1034.193,331.615,372.961,171.898,44.857,158.716
C01242=1034.185,331.368,372.997,171.893,44.855,158.715
C01243=1034.178,331.121,373.032,171.888,44.854,158.714
C01244=1034.170,330.873,373.068,171.882,44.852,158.714
C01245=1034.163,330.626,373.103,171.877,44.852,158.713
C01246=1034.156,330.378,373.139,171.872,44.850,158.712
C01247=1034.149,330.131,373.174,171.867,44.848,158.711
C01248=1034.141,329.884,373.211,171.862,44.847,158.710
C01249=1034.135,329.636,373.246,171.857,44.845,158.709
C01250=1034.127,329.389,373.282,171.852,44.844,158.709
C01251=1034.120,329.141,373.317,171.847,44.842,158.708
C01252=1034.112,328.894,373.353,171.842,44.841,158.707
C01253=1034.106,328.647,373.389,171.837,44.839,158.706
C01254=1034.099,328.399,373.424,171.832,44.838,158.705
C01255=1034.090,328.152,373.459,171.827,44.837,158.704
C01256=1034.084,327.905,373.494,171.821,44.835,158.703
C01257=1034.076,327.657,373.529,171.816,44.834,158.703
C01258=1034.069,327.410,373.564,171.811,44.833,158.702
C01259=1034.061,327.162,373.599,171.806,44.831,158.701
C01260=1034.054,326.915,373.635,171.801,44.830,158.700
C01261=1034.046,326.667,373.670,171.796,44.829,158.700
C01262=1034.039,326.420,373.705,171.791,44.827,158.699
C01263=1034.031,326.173,373.740,171.786,44.826,158.698
C01264=1034.024,325.925,373.775,171.781,44.825,158.697
C01265=1034.016,325.678,373.810,171.776,44.824,158.696
C01266=1034.010,325.430,373.845,171.771,44.822,158.696
C01267=1034.002,325.183,373.880,171.766,44.821,158.695
C01268=1033.995,324.935,373.915,171.761,44.820,158.694
C01269=1033.987,324.688,373.950,171.756,44.819,158.693
C01270=1033.980,324.440,373.985,171.750,44.817,158.692
C01271=1033.972,324.193,374.020,171.746,44.817,158.692
C01272=1033.966,323.946,374.055,171.741,44.815,158.691
C01273=1033.957,323.698,374.090,171.736,44.814,158.690
C01274=1033.951,323.451,374.125,171.731,44.812,158.689
C01275=1033.944,323.203,374.159,171.726,44.812,158.689
C01276=1033.936,322.956,374.193,171.721,44.810,158.688
C01277=1033.929,322.708,374.229,171.716,44.809,158.687
C01278=1033.921,322.461,374.263,171.711,44.807,158.686
C01279=1033.914,322.213,374.298,171.706,44.806,158.686
C01280=1033.907,321.966,374.333,171.701,44.806,158.685
C01281=1033.900,321.718,374.367,171.696,44.804,158.684
C01282=1033.892,321.471,374.402,171.692,44.803,158.683
C01283=1033.881,321.079,374.457,171.684,44.801,158.682
C01284=1033.870,320.686,374.512,171.677,44.799,158.681
C01285=1033.859,320.294,374.567,171.669,44.797,158.680
C01286=1033.848,319.901,374.622,171.661,44.796,158.679
C01287=1033.840,319.654,374.656,171.656,44.795,158.678
C01288=1033.833,319.406,374.692,171.652,44.793,158.677
C01289=1033.826,319.159,374.725,171.647,44.792,158.676
C01290=1033.819,318.911,374.761,171.643,44.791,158.676
C01291=1033.811,318.664,374.795,171.638,44.790,158.675
C01292=1033.804,318.417,374.829,171.633,44.788,158.674
C01293=1033.797,318.169,374.864,171.628,44.788,158.673
C01294=1033.790,317.922,374.898,171.623,44.787,158.673
C01295=1033.783,317.674,374.933,171.618,44.786,158.672
C01296=1033.776,317.427,374.967,171.613,44.784,158.671
C01297=1033.769,317.179,375.002,171.610,44.783,158.671
C01298=1033.762,316.931,375.036,171.605,44.782,158.670
C01299=1033.755,316.684,375.070,171.600,44.781,158.669
C01300=1033.748,316.436,375.105,171.595,44.780,158.669
C01301=1033.741,316.189,375.139,171.590,44.779,158.668
C01302=1033.734,315.941,375.174,171.586,44.778,158.667
C01303=1033.727,315.694,375.208,171.580,44.776,158.666
C01304=1033.720,315.446,375.243,171.577,44.775,158.666
C01305=1033.713,315.199,375.276,171.572,44.774,158.665
C01306=1033.707,314.952,375.310,171.567,44.773,158.664
C01307=1033.700,314.704,375.345,171.562,44.772,158.664
C01308=1033.693,314.457,375.379,171.557,44.771,158.663
C01309=1033.686,314.209,375.413,171.553,44.770,158.662
C01310=1033.679,313.961,375.447,171.549,44.769,158.662
C01311=1033.671,313.714,375.482,171.544,44.768,158.661
C01312=1033.665,313.466,375.516,171.539,44.767,158.660
C01313=1033.658,313.219,375.550,171.535,44.766,158.660
C01314=1033.651,312.971,375.583,171.530,44.765,158.659
C01315=1033.645,312.723,375.618,171.526,44.764,158.658
C01316=1033.637,312.476,375.652,171.521,44.763,158.657
C01317=1033.631,312.228,375.687,171.516,44.762,158.657
C01318=1033.624,311.981,375.720,171.512,44.761,158.656
C01319=1033.617,311.734,375.754,171.508,44.760,158.655
C01320=1033.610,311.486,375.788,171.503,44.759,158.655
C01321=1033.603,311.238,375.822,171.498,44.758,158.654
C01322=1033.595,310.991,375.856,171.493,44.757,158.653
C01323=1033.588,310.743,375.889,171.489,44.757,158.653
C01324=1033.582,310.496,375.923,171.484,44.756,158.652
C01325=1033.574,310.248,375.957,171.480,44.755,158.652
C01326=1033.567,310.000,375.990,171.476,44.754,158.651
C01327=1033.560,309.753,376.023,171.471,44.753,158.650
C01328=1033.552,309.505,376.057,171.466,44.752,158.650
C01329=1033.546,309.258,376.090,171.462,44.752,158.649
C01330=1033.539,309.010,376.124,171.458,44.751,158.648
C01331=1033.531,308.762,376.157,171.453,44.750,158.648
C01332=1033.524,308.515,376.190,171.448,44.750,158.647
C01333=1033.516,308.267,376.224,171.444,44.749,158.647
C01334=1033.510,308.019,376.257,171.439,44.748,158.646
C01335=1033.503,307.772,376.291,171.435,44.747,158.645
C01336=1033.495,307.524,376.324,171.431,44.746,158.645
C01337=1033.489,307.277,376.357,171.426,44.746,158.644
C01338=1033.482,307.029,376.391,171.421,44.745,158.644
C01339=1033.470,306.642,376.443,171.414,44.744,158.643
C01340=1033.459,306.254,376.495,171.408,44.742,158.642
C01341=1033.448,305.867,376.547,171.401,44.741,158.641
C01342=1033.438,305.479,376.599,171.394,44.740,158.640
C01343=1033.430,305.232,376.632,171.389,44.740,158.639
C01344=1033.423,304.984,376.665,171.386,44.738,158.639
C01345=1033.416,304.736,376.699,171.381,44.738,158.638
C01346=1033.409,304.488,376.732,171.376,44.737,158.637
C01347=1033.402,304.241,376.765,171.372,44.737,158.637
C01348=1033.395,303.993,376.798,171.368,44.735,158.636
C01349=1033.389,303.746,376.831,171.363,44.735,158.636
C01350=1033.382,303.498,376.865,171.359,44.735,158.635
C01351=1033.374,303.250,376.897,171.355,44.734,158.635
C01352=1033.367,303.003,376.931,171.351,44.733,158.634
C01353=1033.360,302.755,376.964,171.346,44.732,158.633
C01354=1033.354,302.507,376.996,171.342,44.732,158.633
C01355=1033.346,302.260,377.030,171.337,44.731,158.632
C01356=1033.340,302.012,377.062,171.333,44.730,158.632
C01357=1033.333,301.764,377.095,171.329,44.730,158.631
C01358=1033.326,301.517,377.129,171.325,44.729,158.631
C01359=1033.319,301.269,377.161,171.320,44.728,158.630
C01360=1033.313,301.021,377.194,171.316,44.728,158.630
C01361=1033.305,300.774,377.228,171.312,44.727,158.629
C01362=1033.299,300.526,377.261,171.307,44.726,158.628
C01363=1033.291,300.278,377.293,171.304,44.726,158.628
C01364=1033.285,300.030,377.326,171.299,44.725,158.627
C01365=1033.278,299.782,377.359,171.295,44.724,158.627
C01366=1033.271,299.535,377.392,171.291,44.724,158.626
C01367=1033.265,299.288,377.425,171.286,44.723,158.625
C01368=1033.258,299.040,377.458,171.282,44.722,158.625
C01369=1033.251,298.792,377.491,171.278,44.722,158.624
C01370=1033.244,298.544,377.523,171.273,44.721,158.624
C01371=1033.237,298.296,377.556,171.270,44.720,158.623
C01372=1033.231,298.049,377.589,171.265,44.720,158.623
C01373=1033.224,297.801,377.622,171.261,44.719,158.622
C01374=1033.217,297.554,377.655,171.257,44.718,158.622
C01375=1033.211,297.306,377.687,171.253,44.718,158.621
C01376=1033.204,297.058,377.720,171.249,44.718,158.621
C01377=1033.197,296.811,377.753,171.244,44.717,158.620
C01378=1033.190,296.563,377.785,171.240,44.716,158.619
C01379=1033.184,296.315,377.818,171.236,44.716,158.619
C01380=1033.177,296.067,377.851,171.232,44.715,158.618
C01381=1033.170,295.820,377.883,171.228,44.715,158.618
C01382=1033.163,295.572,377.916,171.224,44.714,158.617
C01383=1033.157,295.323,377.948,171.219,44.713,158.617
C01384=1033.150,295.076,377.981,171.216,44.712,158.616
C01385=1033.143,294.828,378.014,171.211,44.712,158.616
C01386=1033.137,294.580,378.046,171.208,44.712,158.615
C01387=1033.130,294.333,378.079,171.203,44.711,158.615
C01388=1033.123,294.086,378.111,171.199,44.711,158.614
C01389=1033.116,293.837,378.143,171.195,44.710,158.614
C01390=1033.109,293.589,378.175,171.191,44.710,158.613
C01391=1033.102,293.342,378.207,171.187,44.709,158.613
C01392=1033.096,293.094,378.241,171.183,44.709,158.612
C01393=1033.089,292.846,378.272,171.179,44.708,158.612
C01394=1033.083,292.598,378.305,171.174,44.708,158.611
C01395=1033.072,292.228,378.353,171.169,44.707,158.611
C01396=1033.061,291.858,378.400,171.163,44.706,158.610
C01397=1033.051,291.487,378.448,171.156,44.706,158.609
C01398=1033.041,291.117,378.496,171.150,44.706,158.608
C01399=1033.035,290.868,378.528,171.146,44.705,158.608
C01400=1033.027,290.620,378.561,171.142,44.705,158.607
C01401=1033.020,290.372,378.592,171.138,44.704,158.607
C01402=1033.013,290.125,378.624,171.134,44.704,158.606
C01403=1033.007,289.877,378.656,171.130,44.703,158.606
C01404=1033.000,289.629,378.689,171.126,44.703,158.605
C01405=1032.993,289.381,378.720,171.122,44.702,158.605
C01406=1032.986,289.134,378.752,171.118,44.702,158.605
C01407=1032.980,288.886,378.785,171.114,44.702,158.604
C01408=1032.973,288.638,378.816,171.110,44.701,158.604
C01409=1032.966,288.390,378.848,171.106,44.701,158.603
C01410=1032.959,288.142,378.880,171.102,44.700,158.603
C01411=1032.952,287.894,378.912,171.098,44.701,158.602
C01412=1032.945,287.647,378.943,171.094,44.700,158.602
C01413=1032.939,287.398,378.975,171.091,44.699,158.601
C01414=1032.932,287.151,379.008,171.086,44.699,158.601
C01415=1032.925,286.903,379.039,171.083,44.699,158.600
C01416=1032.919,286.655,379.071,171.079,44.699,158.600
C01417=1032.912,286.407,379.102,171.075,44.698,158.599
C01418=1032.904,286.159,379.134,171.071,44.698,158.599
C01419=1032.898,285.911,379.166,171.067,44.698,158.599
C01420=1032.891,285.664,379.197,171.063,44.697,158.598
C01421=1032.884,285.416,379.229,171.059,44.697,158.598
C01422=1032.877,285.168,379.260,171.055,44.697,158.597
C01423=1032.871,284.920,379.292,171.051,44.696,158.597
C01424=1032.864,284.672,379.323,171.047,44.697,158.596
C01425=1032.857,284.424,379.354,171.043,44.696,158.596
C01426=1032.850,284.177,379.387,171.039,44.696,158.596
C01427=1032.843,283.928,379.418,171.036,44.696,158.595
C01428=1032.836,283.680,379.450,171.032,44.695,158.595
C01429=1032.830,283.432,379.481,171.028,44.695,158.594
C01430=1032.823,283.184,379.513,171.024,44.695,158.594
C01431=1032.816,282.937,379.544,171.020,44.695,158.593
C01432=1032.809,282.689,379.575,171.016,44.694,158.593
C01433=1032.802,282.441,379.606,171.012,44.695,158.593
C01434=1032.795,282.193,379.638,171.009,44.694,158.592
C01435=1032.788,281.945,379.669,171.005,44.694,158.592
C01436=1032.782,281.697,379.700,171.001,44.694,158.591
C01437=1032.775,281.449,379.731,170.998,44.694,158.591
C01438=1032.769,281.201,379.763,170.993,44.693,158.591
C01439=1032.762,280.953,379.794,170.989,44.693,158.590
C01440=1032.755,280.705,379.826,170.986,44.693,158.590
C01441=1032.748,280.457,379.857,170.982,44.692,158.589
C01442=1032.742,280.209,379.889,170.978,44.692,158.589
C01443=1032.735,279.961,379.920,170.974,44.692,158.588
C01444=1032.728,279.713,379.951,170.971,44.692,158.588
C01445=1032.722,279.466,379.982,170.967,44.692,158.588
C01446=1032.715,279.218,380.013,170.963,44.692,158.587
C01447=1032.708,278.970,380.044,170.959,44.692,158.587
C01448=1032.701,278.722,380.076,170.956,44.691,158.586
C01449=1032.695,278.474,380.107,170.952,44.691,158.586
C01450=1032.688,278.226,380.138,170.948,44.691,158.586
C01451=1032.679,277.867,380.182,170.943,44.691,158.585
C01452=1032.668,277.509,380.228,170.937,44.690,158.584
C01453=1032.659,277.151,380.273,170.931,44.690,158.584
C01454=1032.649,276.792,380.317,170.926,44.690,158.583
C01455=1032.642,276.544,380.348,170.923,44.690,158.583
C01456=1032.635,276.296,380.379,170.919,44.690,158.583
C01457=1032.630,276.048,380.410,170.915,44.690,158.582
C01458=1032.622,275.800,380.440,170.912,44.690,158.582
C01459=1032.615,275.552,380.472,170.908,44.690,158.582
C01460=1032.609,275.304,380.503,170.904,44.690,158.581
C01461=1032.602,275.056,380.533,170.900,44.690,158.581
C01462=1032.595,274.808,380.564,170.897,44.690,158.580
C01463=1032.588,274.560,380.596,170.893,44.690,158.580
C01464=1032.582,274.312,380.625,170.889,44.689,158.580
C01465=1032.575,274.065,380.657,170.886,44.689,158.579
C01466=1032.569,273.816,380.687,170.882,44.689,158.579
C01467=1032.562,273.568,380.718,170.878,44.689,158.579
C01468=1032.555,273.320,380.749,170.875,44.689,158.578
C01469=1032.548,273.072,380.779,170.871,44.689,158.578
C01470=1032.542,272.824,380.810,170.867,44.689,158.577
C01471=1032.534,272.576,380.840,170.864,44.689,158.577
C01472=1032.528,272.328,380.871,170.860,44.689,158.577
C01473=1032.521,272.080,380.902,170.856,44.689,158.576
C01474=1032.515,271.832,380.932,170.853,44.689,158.576
C01475=1032.508,271.584,380.963,170.850,44.689,158.576
C01476=1032.501,271.336,380.994,170.845,44.689,158.575
C01477=1032.494,271.088,381.025,170.842,44.689,158.575
C01478=1032.488,270.840,381.054,170.839,44.689,158.575
C01479=1032.481,270.592,381.085,170.835,44.689,158.574
C01480=1032.474,270.344,381.116,170.831,44.689,158.574
C01481=1032.468,270.096,381.147,170.828,44.689,158.574
C01482=1032.461,269.848,381.176,170.823,44.689,158.573
C01483=1032.455,269.599,381.207,170.820,44.689,158.573
C01484=1032.447,269.351,381.237,170.817,44.689,158.573
C01485=1032.441,269.104,381.268,170.814,44.689,158.572
C01486=1032.434,268.856,381.298,170.809,44.689,158.572
C01487=1032.427,268.608,381.328,170.806,44.689,158.572
C01488=1032.421,268.359,381.359,170.803,44.689,158.571
C01489=1032.414,268.112,381.389,170.799,44.689,158.571
C01490=1032.408,267.863,381.420,170.795,44.690,158.571
C01491=1032.400,267.615,381.450,170.792,44.690,158.570
C01492=1032.394,267.367,381.480,170.789,44.690,158.570
C01493=1032.387,267.119,381.510,170.785,44.690,158.570
C01494=1032.380,266.871,381.540,170.781,44.690,158.569
C01495=1032.374,266.623,381.571,170.778,44.690,158.569
C01496=1032.367,266.375,381.601,170.774,44.690,158.569
C01497=1032.360,266.126,381.631,170.771,44.690,158.568
C01498=1032.354,265.879,381.661,170.767,44.690,158.568
C01499=1032.347,265.630,381.691,170.764,44.690,158.568
C01500=1032.340,265.382,381.722,170.760,44.690,158.567
C01501=1032.333,265.135,381.751,170.757,44.690,158.567
C01502=1032.326,264.886,381.781,170.753,44.690,158.567
C01503=1032.320,264.639,381.812,170.749,44.690,158.566
C01504=1032.313,264.390,381.842,170.746,44.690,158.566
C01505=1032.306,264.142,381.871,170.743,44.691,158.566
C01506=1032.300,263.894,381.901,170.739,44.691,158.565
C01507=1032.290,263.540,381.944,170.734,44.691,158.565
C01508=1032.281,263.186,381.987,170.729,44.691,158.565
C01509=1032.271,262.832,382.030,170.725,44.692,158.564
C01510=1032.262,262.478,382.072,170.719,44.691,158.564
C01511=1032.255,262.230,382.103,170.716,44.692,158.563
C01512=1032.248,261.983,382.132,170.713,44.692,158.563
C01513=1032.242,261.734,382.163,170.709,44.692,158.563
C01514=1032.236,261.486,382.192,170.705,44.692,158.563
C01515=1032.229,261.238,382.222,170.702,44.692,158.562
C01516=1032.222,260.990,382.252,170.699,44.692,158.562
C01517=1032.215,260.742,382.281,170.696,44.693,158.562
C01518=1032.207,260.494,382.311,170.691,44.693,158.561
C01519=1032.201,260.246,382.340,170.688,44.693,158.561
C01520=1032.194,259.997,382.370,170.685,44.694,158.561
C01521=1032.188,259.749,382.399,170.682,44.694,158.561
C01522=1032.181,259.501,382.429,170.677,44.694,158.560
C01523=1032.174,259.253,382.458,170.674,44.695,158.560
C01524=1032.167,259.005,382.488,170.671,44.695,158.560
C01525=1032.160,258.757,382.517,170.668,44.695,158.560
C01526=1032.153,258.509,382.547,170.665,44.696,158.559
C01527=1032.146,258.260,382.576,170.661,44.696,158.559
C01528=1032.140,258.012,382.606,170.657,44.696,158.559
C01529=1032.133,257.763,382.636,170.654,44.696,158.559
C01530=1032.126,257.516,382.665,170.651,44.696,158.558
C01531=1032.119,257.267,382.694,170.648,44.697,158.558
C01532=1032.112,257.019,382.723,170.644,44.697,158.558
C01533=1032.105,256.771,382.753,170.640,44.697,158.557
C01534=1032.099,256.523,382.782,170.637,44.698,158.557
C01535=1032.092,256.274,382.812,170.634,44.698,158.557
C01536=1032.085,256.027,382.841,170.631,44.698,158.557
C01537=1032.079,255.779,382.870,170.628,44.699,158.556
C01538=1032.072,255.530,382.899,170.623,44.699,158.556
C01539=1032.065,255.282,382.929,170.620,44.700,158.556
C01540=1032.058,255.034,382.958,170.617,44.700,158.556
C01541=1032.052,254.785,382.988,170.614,44.700,158.555
C01542=1032.045,254.537,383.018,170.611,44.700,158.555
C01543=1032.038,254.289,383.046,170.607,44.700,158.555
C01544=1032.032,254.041,383.075,170.603,44.701,158.555
C01545=1032.024,253.793,383.105,170.600,44.701,158.554
C01546=1032.018,253.545,383.134,170.597,44.702,158.554
C01547=1032.011,253.296,383.164,170.594,44.702,158.554
C01548=1032.005,253.048,383.193,170.591,44.702,158.554
C01549=1031.998,252.800,383.221,170.588,44.702,158.553
C01550=1031.991,252.552,383.251,170.584,44.703,158.553
C01551=1031.985,252.304,383.280,170.581,44.703,158.553
C01552=1031.978,252.055,383.310,170.577,44.703,158.553
C01553=1031.972,251.807,383.339,170.574,44.704,158.552
C01554=1031.965,251.559,383.367,170.571,44.704,158.552
C01555=1031.958,251.310,383.397,170.568,44.705,158.552
C01556=1031.951,251.063,383.426,170.564,44.705,158.552
C01557=1031.945,250.815,383.455,170.561,44.705,158.551
C01558=1031.938,250.566,383.485,170.558,44.705,158.551
C01559=1031.931,250.318,383.513,170.555,44.705,158.551
C01560=1031.925,250.070,383.542,170.552,44.706,158.551
C01561=1031.919,249.822,383.571,170.548,44.706,158.550
C01562=1031.912,249.573,383.601,170.545,44.707,158.550
C01563=1031.902,249.217,383.643,170.540,44.707,158.550
C01564=1031.893,248.863,383.684,170.536,44.707,158.549
C01565=1031.884,248.507,383.725,170.531,44.708,158.549
C01566=1031.874,248.152,383.767,170.526,44.709,158.549
C01567=1031.867,247.904,383.796,170.523,44.709,158.549
C01568=1031.861,247.656,383.825,170.520,44.709,158.548
C01569=1031.855,247.408,383.854,170.517,44.709,158.548
C01570=1031.848,247.159,383.883,170.514,44.710,158.548
C01571=1031.842,246.911,383.912,170.511,44.711,158.548
C01572=1031.835,246.663,383.941,170.507,44.711,158.547
C01573=1031.828,246.415,383.970,170.504,44.711,158.547
C01574=1031.822,246.166,383.999,170.501,44.711,158.547
C01575=1031.815,245.918,384.028,170.498,44.712,158.547
C01576=1031.809,245.670,384.057,170.495,44.712,158.547
C01577=1031.802,245.422,384.086,170.492,44.713,158.546
C01578=1031.796,245.173,384.114,170.488,44.713,158.546
C01579=1031.790,244.925,384.143,170.485,44.713,158.546
C01580=1031.783,244.676,384.172,170.482,44.713,158.546
C01581=1031.776,244.428,384.201,170.479,44.714,158.545
C01582=1031.770,244.180,384.230,170.475,44.715,158.545
C01583=1031.763,243.932,384.258,170.472,44.715,158.545
C01584=1031.757,243.684,384.287,170.469,44.715,158.545
C01585=1031.751,243.435,384.316,170.466,44.716,158.545
C01586=1031.743,243.187,384.345,170.462,44.716,158.544
C01587=1031.737,242.938,384.373,170.459,44.717,158.544
C01588=1031.730,242.690,384.401,170.456,44.717,158.544
C01589=1031.724,242.442,384.430,170.453,44.717,158.544
C01590=1031.717,242.194,384.458,170.450,44.718,158.544
C01591=1031.711,241.946,384.487,170.447,44.719,158.543
C01592=1031.703,241.697,384.516,170.444,44.719,158.543
C01593=1031.697,241.448,384.544,170.441,44.719,158.543
C01594=1031.690,241.201,384.573,170.438,44.720,158.543
C01595=1031.684,240.952,384.602,170.435,44.721,158.543
C01596=1031.677,240.704,384.630,170.431,44.721,158.542
C01597=1031.671,240.456,384.659,170.428,44.721,158.542
C01598=1031.665,240.207,384.686,170.425,44.722,158.542
C01599=1031.657,239.959,384.715,170.422,44.723,158.542
C01600=1031.651,239.710,384.743,170.419,44.723,158.542
C01601=1031.644,239.462,384.772,170.416,44.723,158.541
C01602=1031.637,239.214,384.800,170.413,44.724,158.541
C01603=1031.630,238.966,384.828,170.410,44.725,158.541
C01604=1031.624,238.717,384.856,170.407,44.725,158.541
C01605=1031.617,238.469,384.885,170.404,44.726,158.541
C01606=1031.611,238.221,384.913,170.400,44.726,158.540
C01607=1031.603,237.972,384.941,170.397,44.727,158.540
C01608=1031.597,237.724,384.970,170.394,44.727,158.540
C01609=1031.591,237.475,384.997,170.391,44.728,158.540
C01610=1031.584,237.227,385.026,170.388,44.728,158.540
C01611=1031.577,236.979,385.054,170.385,44.729,158.540
C01612=1031.571,236.731,385.083,170.382,44.730,158.540
C01613=1031.564,236.482,385.110,170.379,44.730,158.539
C01614=1031.557,236.234,385.138,170.376,44.730,158.539
C01615=1031.550,235.986,385.167,170.373,44.731,158.539
C01616=1031.544,235.738,385.194,170.370,44.732,158.539
C01617=1031.538,235.489,385.223,170.367,44.732,158.539
C01618=1031.531,235.241,385.250,170.364,44.733,158.538
C01619=1031.521,234.880,385.291,170.360,44.734,158.538
C01620=1031.511,234.518,385.332,170.356,44.735,158.538
C01621=1031.501,234.157,385.373,170.351,44.736,158.538
C01622=1031.491,233.795,385.413,170.346,44.736,158.537
C01623=1031.485,233.547,385.442,170.343,44.737,158.537
C01624=1031.478,233.299,385.470,170.340,44.737,158.537
C01625=1031.472,233.050,385.498,170.337,44.738,158.537
C01626=1031.465,232.802,385.526,170.334,44.739,158.537
C01627=1031.459,232.554,385.553,170.331,44.739,158.537
C01628=1031.452,232.306,385.581,170.328,44.740,158.536
C01629=1031.446,232.058,385.610,170.325,44.741,158.536
C01630=1031.439,231.809,385.637,170.322,44.741,158.536
C01631=1031.433,231.561,385.665,170.319,44.742,158.536
C01632=1031.426,231.312,385.693,170.316,44.743,158.536
C01633=1031.419,231.064,385.721,170.314,44.743,158.536
C01634=1031.413,230.815,385.748,170.311,44.744,158.536
C01635=1031.406,230.567,385.776,170.308,44.744,158.535
C01636=1031.399,230.319,385.805,170.305,44.745,158.535
C01637=1031.392,230.071,385.832,170.302,44.746,158.535
C01638=1031.386,229.822,385.860,170.299,44.746,158.535
C01639=1031.379,229.574,385.888,170.296,44.747,158.535
C01640=1031.372,229.325,385.915,170.293,44.747,158.535
C01641=1031.366,229.077,385.943,170.290,44.748,158.534
C01642=1031.359,228.829,385.971,170.287,44.749,158.534
C01643=1031.352,228.580,385.999,170.284,44.749,158.534
C01644=1031.346,228.332,386.026,170.281,44.750,158.534
C01645=1031.339,228.084,386.054,170.277,44.751,158.534
C01646=1031.333,227.836,386.081,170.275,44.751,158.534
C01647=1031.326,227.586,386.108,170.272,44.752,158.534
C01648=1031.320,227.338,386.136,170.269,44.752,158.533
C01649=1031.313,227.090,386.164,170.266,44.753,158.533
C01650=1031.306,226.841,386.192,170.264,44.754,158.533
C01651=1031.299,226.593,386.219,170.261,44.755,158.533
C01652=1031.292,226.345,386.247,170.257,44.756,158.533
C01653=1031.286,226.096,386.274,170.254,44.756,158.533
C01654=1031.279,225.847,386.301,170.251,44.757,158.533
C01655=1031.273,225.599,386.329,170.248,44.758,158.532
C01656=1031.266,225.351,386.356,170.246,44.759,158.533
C01657=1031.259,225.103,386.384,170.243,44.760,158.532
C01658=1031.253,224.854,386.411,170.239,44.760,158.532
C01659=1031.246,224.605,386.438,170.237,44.761,158.532
C01660=1031.239,224.357,386.465,170.234,44.761,158.532
C01661=1031.232,224.109,386.493,170.231,44.762,158.532
C01662=1031.226,223.860,386.520,170.229,44.763,158.532
C01663=1031.219,223.612,386.547,170.226,44.764,158.532
C01664=1031.213,223.363,386.575,170.223,44.764,158.531
C01665=1031.205,223.115,386.602,170.219,44.765,158.531
C01666=1031.199,222.866,386.629,170.216,44.766,158.531
C01667=1031.192,222.618,386.657,170.213,44.766,158.531
C01668=1031.186,222.370,386.684,170.212,44.768,158.531
C01669=1031.179,222.121,386.711,170.209,44.768,158.531
C01670=1031.172,221.873,386.739,170.206,44.769,158.531
C01671=1031.166,221.624,386.766,170.203,44.769,158.531
C01672=1031.159,221.375,386.793,170.199,44.770,158.530
C01673=1031.153,221.128,386.820,170.197,44.771,158.530
C01674=1031.146,220.880,386.848,170.194,44.772,158.530
C01675=1031.136,220.511,386.888,170.190,44.773,158.530
C01676=1031.126,220.141,386.929,170.186,44.774,158.530
C01677=1031.117,219.772,386.969,170.182,44.775,158.530
C01678=1031.107,219.404,387.010,170.177,44.776,158.530
C01679=1031.100,219.155,387.037,170.175,44.777,158.529
C01680=1031.093,218.908,387.063,170.172,44.778,158.529
C01681=1031.087,218.659,387.090,170.169,44.779,158.529
C01682=1031.080,218.410,387.117,170.166,44.779,158.529
C01683=1031.073,218.161,387.145,170.163,44.781,158.529
C01684=1031.067,217.913,387.171,170.160,44.781,158.529
C01685=1031.060,217.665,387.198,170.157,44.782,158.529
C01686=1031.053,217.416,387.225,170.155,44.783,158.529
C01687=1031.046,217.168,387.252,170.152,44.784,158.529
C01688=1031.040,216.920,387.279,170.149,44.784,158.529
C01689=1031.033,216.671,387.306,170.146,44.786,158.529
C01690=1031.026,216.422,387.333,170.143,44.786,158.528
C01691=1031.020,216.173,387.360,170.140,44.787,158.528
C01692=1031.013,215.925,387.386,170.137,44.788,158.528
C01693=1031.006,215.677,387.413,170.135,44.789,158.528
C01694=1030.999,215.428,387.440,170.133,44.790,158.528
C01695=1030.993,215.180,387.467,170.130,44.791,158.528
C01696=1030.986,214.932,387.494,170.127,44.791,158.528
C01697=1030.979,214.683,387.520,170.124,44.792,158.528
C01698=1030.973,214.434,387.547,170.121,44.793,158.528
C01699=1030.966,214.186,387.574,170.119,44.794,158.528
C01700=1030.959,213.937,387.601,170.116,44.795,158.528
C01701=1030.952,213.689,387.627,170.113,44.796,158.527
C01702=1030.946,213.441,387.655,170.110,44.796,158.527
C01703=1030.939,213.192,387.681,170.107,44.797,158.527
C01704=1030.933,212.944,387.708,170.105,44.798,158.527
C01705=1030.926,212.695,387.734,170.102,44.799,158.527
C01706=1030.919,212.447,387.762,170.099,44.800,158.527
C01707=1030.913,212.198,387.788,170.096,44.800,158.527
C01708=1030.907,211.949,387.815,170.093,44.802,158.527
C01709=1030.899,211.701,387.841,170.091,44.802,158.527
C01710=1030.894,211.452,387.868,170.088,44.803,158.527
C01711=1030.886,211.204,387.895,170.086,44.804,158.527
C01712=1030.880,210.956,387.921,170.082,44.805,158.526
C01713=1030.873,210.707,387.948,170.080,44.806,158.526
C01714=1030.866,210.458,387.975,170.078,44.806,158.526
C01715=1030.860,210.210,388.001,170.075,44.808,158.526
C01716=1030.853,209.961,388.028,170.072,44.808,158.526
C01717=1030.846,209.712,388.054,170.069,44.810,158.526
C01718=1030.839,209.465,388.081,170.066,44.810,158.526
C01719=1030.832,209.216,388.107,170.064,44.811,158.526
C01720=1030.827,208.968,388.134,170.061,44.812,158.526
C01721=1030.819,208.719,388.160,170.058,44.813,158.526
C01722=1030.812,208.470,388.187,170.055,44.814,158.526
C01723=1030.807,208.222,388.213,170.053,44.814,158.526
C01724=1030.799,207.973,388.240,170.051,44.816,158.526
C01725=1030.793,207.725,388.266,170.048,44.817,158.526
C01726=1030.786,207.477,388.292,170.045,44.818,158.525
C01727=1030.779,207.228,388.318,170.042,44.819,158.525
C01728=1030.773,206.979,388.345,170.040,44.819,158.525
C01729=1030.766,206.731,388.372,170.037,44.821,158.525
C01730=1030.759,206.483,388.398,170.034,44.821,158.525
C01731=1030.750,206.119,388.436,170.030,44.823,158.525
C01732=1030.739,205.756,388.474,170.026,44.824,158.525
C01733=1030.729,205.394,388.513,170.023,44.826,158.525
C01734=1030.720,205.031,388.550,170.019,44.827,158.525
C01735=1030.694,203.981,388.656,169.664,44.724,158.469
C01736=1030.688,203.733,388.681,169.660,44.725,158.469
C01737=1030.683,203.484,388.705,169.657,44.727,158.469
C01738=1030.676,203.235,388.731,169.653,44.729,158.469
C01739=1030.670,202.988,388.755,169.650,44.730,158.469
C01740=1030.664,202.738,388.780,169.646,44.732,158.469
C01741=1030.658,202.490,388.805,169.643,44.734,158.469
C01742=1030.652,202.240,388.830,169.639,44.735,158.469
C01743=1030.646,201.992,388.855,169.635,44.737,158.469
C01744=1030.641,201.743,388.879,169.632,44.739,158.469
C01745=1030.634,201.495,388.904,169.628,44.740,158.469
C01746=1030.628,201.246,388.928,169.624,44.743,158.469
C01747=1030.622,200.998,388.954,169.620,44.744,158.469
C01748=1030.616,200.748,388.978,169.617,44.746,158.469
C01749=1030.611,200.500,389.003,169.613,44.748,158.469
C01750=1030.605,200.251,389.028,169.610,44.750,158.469
C01751=1030.598,200.002,389.052,169.606,44.751,158.469
C01752=1030.592,199.754,389.077,169.602,44.753,158.469
C01753=1030.586,199.505,389.101,169.599,44.755,158.469
C01754=1030.579,199.256,389.125,169.596,44.757,158.469
C01755=1030.574,199.008,389.150,169.592,44.759,158.469
C01756=1030.567,198.759,389.174,169.588,44.761,158.469
C01757=1030.561,198.510,389.199,169.585,44.763,158.469
C01758=1030.555,198.262,389.222,169.581,44.765,158.469
C01759=1030.549,198.013,389.248,169.577,44.766,158.469
C01760=1030.542,197.764,389.272,169.574,44.769,158.469
C01761=1030.537,197.515,389.296,169.570,44.770,158.469
C01762=1030.530,197.266,389.320,169.567,44.772,158.469
C01763=1030.524,197.017,389.344,169.563,44.774,158.469
C01764=1030.518,196.769,389.369,169.559,44.776,158.469
C01765=1030.512,196.520,389.393,169.556,44.778,158.470
C01766=1030.506,196.272,389.417,169.553,44.780,158.470
C01767=1030.500,196.023,389.442,169.549,44.781,158.470
C01768=1030.493,195.774,389.466,169.546,44.784,158.470
C01769=1030.488,195.525,389.490,169.542,44.786,158.470
C01770=1030.481,195.277,389.515,169.538,44.787,158.470
C01771=1030.476,195.028,389.539,169.535,44.789,158.470
C01772=1030.469,194.779,389.563,169.531,44.792,158.470
C01773=1030.464,194.530,389.587,169.527,44.793,158.470
C01774=1030.457,194.282,389.611,169.525,44.795,158.470
C01775=1030.451,194.032,389.636,169.521,44.797,158.470
C01776=1030.445,193.784,389.660,169.517,44.799,158.470
C01777=1030.440,193.535,389.684,169.514,44.801,158.470
C01778=1030.433,193.286,389.708,169.510,44.803,158.470
C01779=1030.427,193.037,389.732,169.506,44.804,158.470
C01780=1030.422,192.789,389.756,169.503,44.807,158.470
C01781=1030.415,192.540,389.780,169.500,44.809,158.470
C01782=1030.410,192.291,389.804,169.497,44.811,158.470
C01783=1030.403,192.042,389.829,169.493,44.812,158.470
C01784=1030.398,191.794,389.853,169.489,44.814,158.471
C01785=1030.391,191.545,389.877,169.486,44.817,158.471
C01786=1030.386,191.296,389.901,169.483,44.818,158.471
C01787=1030.380,191.048,389.925,169.479,44.820,158.471
C01788=1030.374,190.799,389.949,169.476,44.822,158.471
C01789=1030.368,190.550,389.973,169.472,44.824,158.471
C01790=1030.361,190.301,389.997,169.469,44.826,158.471
C01791=1030.356,190.053,390.021,169.466,44.828,158.471
C01792=1030.349,189.804,390.045,169.462,44.830,158.471
C01793=1030.344,189.555,390.070,169.459,44.831,158.471
C01794=1030.338,189.306,390.093,169.455,44.834,158.471
C01795=1030.332,189.057,390.117,169.451,44.836,158.471
C01796=1030.325,188.774,390.144,169.448,44.838,158.471
C01797=1030.319,188.491,390.172,169.444,44.840,158.471
C01798=1030.312,188.207,390.199,169.441,44.842,158.471
C01799=1030.305,187.923,390.226,169.436,44.845,158.471
C01800=1030.299,187.675,390.250,169.433,44.847,158.472
C01801=1030.293,187.426,390.275,169.430,44.848,158.472
C01802=1030.288,187.177,390.298,169.426,44.850,158.472
C01803=1030.282,186.929,390.321,169.423,44.852,158.472
C01804=1030.276,186.679,390.346,169.420,44.854,158.472
C01805=1030.270,186.431,390.369,169.416,44.856,158.472
C01806=1030.264,186.182,390.394,169.413,44.858,158.472
C01807=1030.258,185.933,390.417,169.409,44.860,158.472
C01808=1030.252,185.685,390.441,169.407,44.862,158.472
C01809=1030.247,185.436,390.465,169.403,44.864,158.472
